KUKA KRL program: MyProgram_224().src

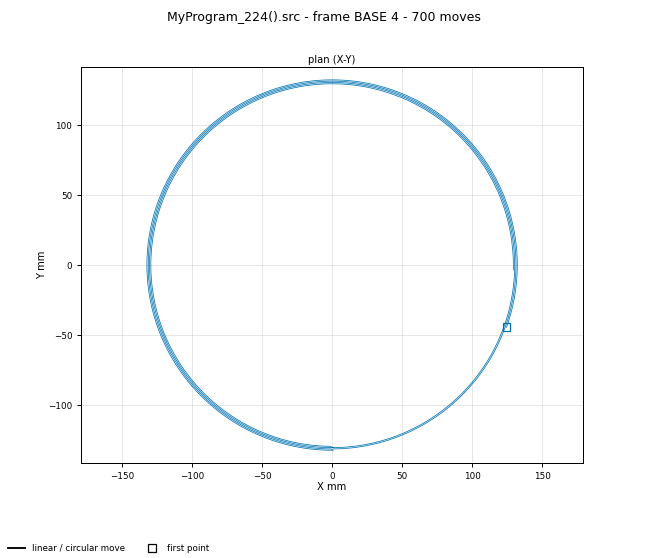
[picture p0: tool path of MyProgram_224().src in frame BASE 4, 700 of 700 moves have a stored position in this frame; points joined in program order, loops and branches not executed]
&ACCESS RVP
&REL 1
&PARAM TEMPLATE = C:\KRC\Roboter\Template\vorgabe
&PARAM EDITMASK = *
DEF MyProgram_224()
; ---- Setting reference (Base) ----
$BASE = BASE_DATA[4]

; --------------------------
; ---- Setting tool (TCP) ----
$TOOL = TOOL_DATA[3]
; --------------------------

$VEL.CP = VEL_APROX_PRINT
Startdeposition()
$VEL.CP = VEL_PRINT
LIN {X 124.5502,Y -44.5049,Z 155,A -21.604,B 21.391,C -0.8343,E1 21.5573,E2 829.1643} C_DIS
LIN {X 125.729,Y -41.0623,Z 155,A -19.4194,B 21.3896,C -0.8684,E1 21.5593,E2 826.9015} C_DIS
LIN {X 127.1456,Y -36.4403,Z 155,A -17.9667,B 21.3906,C -0.844,E1 21.5603,E2 825.525} C_DIS
LIN {X 127.8136,Y -34.0149,Z 155,A -16.9109,B 21.3905,C -0.8459,E1 21.5611,E2 824.4715} C_DIS
LIN {X 128.5807,Y -30.9894,Z 155,A -15.17,B 21.3896,C -0.8688,E1 21.5623,E2 822.6801} C_DIS
LIN {X 129.3697,Y -27.5135,Z 155,A -14.0813,B 21.3903,C -0.8518,E1 21.5629,E2 821.6452} C_DIS
LIN {X 129.9607,Y -24.5693,Z 155,A -12.5854,B 21.3897,C -0.8653,E1 21.5637,E2 820.123} C_DIS
LIN {X 130.7,Y -20.2702,Z 155,A -10.8405,B 21.3897,C -0.8643,E1 21.5645,E2 818.3928} C_DIS
LIN {X 131.174,Y -16.9359,Z 155,A -9.3618,B 21.3896,C -0.8699,E1 21.565,E2 816.9092} C_DIS
LIN {X 131.7113,Y -12.0763,Z 155,A -7.3959,B 21.3896,C -0.8694,E1 21.5656,E2 814.9586} C_DIS
LIN {X 132.0248,Y -7.9307,Z 155,A -5.4229,B 21.389,C -0.8834,E1 21.566,E2 812.9614} C_DIS
LIN {X 132.2116,Y -3.6774,Z 155,A -3.6274,B 21.3889,C -0.8869,E1 21.5662,E2 811.1688} C_DIS
LIN {X 132.263,Y 0.4651,Z 155,A -1.8131,B 21.3886,C -0.8936,E1 21.5662,E2 809.3493} C_DIS
LIN {X 132.2015,Y 4.0385,Z 155,A -0.2395,B 21.3884,C -0.8998,E1 21.5661,E2 807.7701} C_DIS
LIN {X 132.0289,Y 7.8652,Z 155,A 1.3524,B 21.3884,C -0.9018,E1 21.5659,E2 806.1838} C_DIS
LIN {X 131.7496,Y 11.6494,Z 155,A 3.0747,B 21.3879,C -0.9108,E1 21.5655,E2 804.4493} C_DIS
LIN {X 131.3233,Y 15.7351,Z 155,A 4.5909,B 21.3882,C -0.9038,E1 21.565,E2 802.9627} C_DIS
LIN {X 130.9162,Y 18.8242,Z 155,A 5.9988,B 21.3879,C -0.9108,E1 21.5645,E2 801.5455} C_DIS
LIN {X 130.4526,Y 21.8058,Z 155,A 7.3862,B 21.3876,C -0.9187,E1 21.5638,E2 800.1463} C_DIS
LIN {X 129.5637,Y 26.583,Z 155,A 10.6351,B 21.385,C -0.9803,E1 21.562,E2 796.7521} C_DIS
LIN {X 127.7263,Y 34.3422,Z 155,A 12.4336,B 21.3879,C -0.9114,E1 21.5609,E2 795.1537} C_DIS
LIN {X 126.694,Y 37.9805,Z 155,A 14.4558,B 21.387,C -0.9345,E1 21.5593,E2 793.0824} C_DIS
LIN {X 125.6249,Y 41.3749,Z 155,A 16.0763,B 21.3866,C -0.9428,E1 21.5578,E2 791.45} C_DIS
LIN {X 124.4093,Y 44.8959,Z 155,A 17.6313,B 21.3866,C -0.9448,E1 21.5564,E2 789.9} C_DIS
LIN {X 123.2107,Y 48.088,Z 155,A 19.0995,B 21.3864,C -0.9487,E1 21.5549,E2 788.4309} C_DIS
LIN {X 121.8494,Y 51.442,Z 155,A 20.6359,B 21.3862,C -0.9517,E1 21.5533,E2 786.8964} C_DIS
LIN {X 120.5815,Y 54.3464,Z 155,A 22.5754,B 21.3849,C -0.9825,E1 21.551,E2 784.8854} C_DIS
LIN {X 118.6107,Y 58.5216,Z 155,A 23.667,B 21.3865,C -0.9451,E1 21.5498,E2 783.9027} C_DIS
LIN {X 117.3355,Y 61.0402,Z 155,A 25.0814,B 21.386,C -0.9575,E1 21.548,E2 782.4636} C_DIS
LIN {X 115.8159,Y 63.8789,Z 155,A 26.7141,B 21.3854,C -0.9724,E1 21.5457,E2 780.8003} C_DIS
LIN {X 113.4513,Y 67.9904,Z 155,A 28.7424,B 21.3852,C -0.9767,E1 21.5429,E2 778.7729} C_DIS
LIN {X 111.1551,Y 71.6833,Z 155,A 30.6297,B 21.385,C -0.9817,E1 21.54,E2 776.8831} C_DIS
LIN {X 108.7622,Y 75.2641,Z 155,A 32.5525,B 21.3846,C -0.9892,E1 21.537,E2 774.9513} C_DIS
LIN {X 106.7868,Y 78.0415,Z 155,A 33.9503,B 21.3846,C -0.9892,E1 21.5347,E2 773.5616} C_DIS
LIN {X 104.1105,Y 81.5771,Z 155,A 36.6611,B 21.3827,C -1.031,E1 21.5299,E2 770.7518} C_DIS
LIN {X 99.9718,Y 86.6001,Z 155,A 38.3531,B 21.3848,C -0.9846,E1 21.5271,E2 769.1956} C_DIS
LIN {X 96.5456,Y 90.404,Z 155,A 40.8663,B 21.384,C -1.0033,E1 21.5223,E2 766.6446} C_DIS
LIN {X 93.4654,Y 93.5849,Z 155,A 42.7806,B 21.3838,C -1.0072,E1 21.5185,E2 764.7292} C_DIS
LIN {X 86.4701,Y 100.0837,Z 155,A 46.5284,B 21.3843,C -0.9976,E1 21.5109,E2 761.0258} C_DIS
LIN {X 83.7881,Y 102.3395,Z 155,A 48.3808,B 21.3834,C -1.0159,E1 21.5068,E2 759.132} C_DIS
LIN {X 80.2289,Y 105.1529,Z 155,A 50.3468,B 21.3833,C -1.0195,E1 21.5025,E2 757.1647} C_DIS
LIN {X 76.5729,Y 107.845,Z 155,A 52.3369,B 21.3831,C -1.024,E1 21.498,E2 755.1707} C_DIS
LIN {X 72.8868,Y 110.3692,Z 155,A 54.236,B 21.383,C -1.0255,E1 21.4936,E2 753.2751} C_DIS
LIN {X 68.9512,Y 112.8698,Z 155,A 56.2434,B 21.3829,C -1.028,E1 21.4888,E2 751.2683} C_DIS
LIN {X 64.7177,Y 115.3492,Z 155,A 58.3316,B 21.3829,C -1.0294,E1 21.4838,E2 749.1838} C_DIS
LIN {X 60.9874,Y 117.3632,Z 155,A 60.4088,B 21.3822,C -1.0429,E1 21.4786,E2 747.0768} C_DIS
LIN {X 57.9889,Y 118.8735,Z 155,A 61.7981,B 21.3822,C -1.0417,E1 21.4751,E2 745.695} C_DIS
LIN {X 53.656,Y 120.8903,Z 155,A 63.5823,B 21.3827,C -1.0312,E1 21.4707,E2 743.9449} C_DIS
LIN {X 51.011,Y 122.0294,Z 155,A 64.8174,B 21.3827,C -1.032,E1 21.4675,E2 742.7111} C_DIS
LIN {X 47.2563,Y 123.534,Z 155,A 66.535,B 21.3827,C -1.0322,E1 21.463,E2 740.9976} C_DIS
LIN {X 43.2481,Y 124.9917,Z 155,A 68.4763,B 21.3824,C -1.0381,E1 21.4579,E2 739.0447} C_DIS
LIN {X 39.7093,Y 126.1618,Z 155,A 70.0332,B 21.3824,C -1.0368,E1 21.4538,E2 737.4948} C_DIS
LIN {X 33.5194,Y 127.9458,Z 155,A 73.1745,B 21.3816,C -1.0545,E1 21.4452,E2 734.3114} C_DIS
LIN {X 30.1368,Y 128.7851,Z 155,A 74.2876,B 21.3824,C -1.0376,E1 21.4423,E2 733.2463} C_DIS
LIN {X 26.5128,Y 129.578,Z 155,A 75.9495,B 21.3823,C -1.0409,E1 21.4378,E2 731.578} C_DIS
LIN {X 23.2374,Y 130.2052,Z 155,A 77.392,B 21.3823,C -1.0414,E1 21.4338,E2 730.136} C_DIS
LIN {X 19.5153,Y 130.8169,Z 155,A 79.2255,B 21.3818,C -1.0507,E1 21.4287,E2 728.2789} C_DIS
LIN {X 15.5547,Y 131.3448,Z 155,A 80.7732,B 21.3822,C -1.0431,E1 21.4245,E2 726.7537} C_DIS
LIN {X 11.8097,Y 131.7361,Z 155,A 82.5091,B 21.382,C -1.0479,E1 21.4196,E2 725.0059} C_DIS
LIN {X 7.9894,Y 132.0212,Z 155,A 84.0684,B 21.3822,C -1.0436,E1 21.4153,E2 723.4592} C_DIS
LIN {X 3.5658,Y 132.2147,Z 155,A 85.9886,B 21.3822,C -1.0436,E1 21.4099,E2 721.5397} C_DIS
LIN {X -0.6478,Y 132.2612,Z 155,A 87.8269,B 21.3822,C -1.0439,E1 21.4048,E2 719.7007} C_DIS
LIN {X -4.8887,Y 132.1726,Z 155,A 89.6565,B 21.3822,C -1.0431,E1 21.3997,E2 717.873} C_DIS
LIN {X -8.5001,Y 131.9898,Z 155,A 91.3658,B 21.3819,C -1.0488,E1 21.3949,E2 716.1475} C_DIS
LIN {X -13.2402,Y 131.5996,Z 155,A 93.3984,B 21.382,C -1.0466,E1 21.3893,E2 714.1196} C_DIS
LIN {X -17.2614,Y 131.1314,Z 155,A 95.0131,B 21.3823,C -1.0396,E1 21.3848,E2 712.5227} C_DIS
LIN {X -21.0472,Y 130.5792,Z 155,A 97.0435,B 21.3816,C -1.0547,E1 21.3791,E2 710.4488} C_DIS
LIN {X -24.4702,Y 129.9796,Z 155,A 98,B 21.3828,C -1.0299,E1 21.3767,E2 709.5592} C_DIS
LIN {X -26.9614,Y 129.4867,Z 155,A 100.1971,B 21.3806,C -1.0765,E1 21.3703,E2 707.231} C_DIS
LIN {X -33.2052,Y 128.0282,Z 155,A 102.0517,B 21.3826,C -1.0339,E1 21.3656,E2 705.4902} C_DIS
LIN {X -38.8586,Y 126.4253,Z 155,A 104.581,B 21.3828,C -1.0306,E1 21.3588,E2 702.9652} C_DIS
LIN {X -41.9806,Y 125.4232,Z 155,A 106.0925,B 21.3827,C -1.0328,E1 21.3548,E2 701.4443} C_DIS
LIN {X -45.4039,Y 124.2261,Z 155,A 107.7019,B 21.3827,C -1.0325,E1 21.3505,E2 699.8319} C_DIS
LIN {X -54.3042,Y 120.6004,Z 155,A 111.6937,B 21.3833,C -1.0194,E1 21.3403,E2 695.8653} C_DIS
LIN {X -56.8154,Y 119.4376,Z 155,A 113.5157,B 21.3821,C -1.0441,E1 21.3355,E2 693.97} C_DIS
LIN {X -60.8021,Y 117.4605,Z 155,A 115.0137,B 21.3831,C -1.0227,E1 21.3319,E2 692.526} C_DIS
LIN {X -64.4819,Y 115.4817,Z 155,A 116.8834,B 21.3831,C -1.0222,E1 21.3274,E2 690.6514} C_DIS
LIN {X -68.3799,Y 113.2166,Z 155,A 118.7978,B 21.3834,C -1.0171,E1 21.3228,E2 688.744} C_DIS
LIN {X -72.1535,Y 110.8499,Z 155,A 120.7581,B 21.3834,C -1.0149,E1 21.3182,E2 686.7825} C_DIS
LIN {X -75.9078,Y 108.3142,Z 155,A 122.7343,B 21.3836,C -1.0116,E1 21.3136,E2 684.8073} C_DIS
LIN {X -79.3536,Y 105.8157,Z 155,A 124.6149,B 21.3837,C -1.0094,E1 21.3094,E2 682.9248} C_DIS
LIN {X -82.9748,Y 102.9999,Z 155,A 126.5719,B 21.384,C -1.004,E1 21.3051,E2 680.9742} C_DIS
LIN {X -86.4303,Y 100.118,Z 155,A 128.5306,B 21.3841,C -1.0001,E1 21.3009,E2 679.017} C_DIS
LIN {X -89.4659,Y 97.4148,Z 155,A 130.2762,B 21.3843,C -0.9955,E1 21.2973,E2 677.2759} C_DIS
LIN {X -92.5632,Y 94.4767,Z 155,A 132.184,B 21.3844,C -0.9936,E1 21.2935,E2 675.3638} C_DIS
LIN {X -95.8388,Y 91.1527,Z 155,A 134.2016,B 21.3846,C -0.9886,E1 21.2896,E2 673.3497} C_DIS
LIN {X -98.8107,Y 87.9227,Z 155,A 136.1481,B 21.3848,C -0.9858,E1 21.2859,E2 671.4007} C_DIS
LIN {X -101.7408,Y 84.5141,Z 155,A 138.0878,B 21.385,C -0.9805,E1 21.2825,E2 669.4649} C_DIS
LIN {X -104.624,Y 80.9174,Z 155,A 140.0687,B 21.3853,C -0.9746,E1 21.279,E2 667.4892} C_DIS
LIN {X -107.2983,Y 77.3369,Z 155,A 142.0449,B 21.3854,C -0.9711,E1 21.2758,E2 665.5112} C_DIS
LIN {X -109.7964,Y 73.7475,Z 155,A 143.9683,B 21.3856,C -0.9672,E1 21.2727,E2 663.5874} C_DIS
LIN {X -112.3661,Y 69.7687,Z 155,A 145.9858,B 21.3859,C -0.9601,E1 21.2697,E2 661.5774} C_DIS
LIN {X -114.6205,Y 66.0003,Z 155,A 147.9225,B 21.3861,C -0.9561,E1 21.267,E2 659.6397} C_DIS
LIN {X -116.7267,Y 62.1995,Z 155,A 149.701,B 21.3865,C -0.9464,E1 21.2646,E2 657.8766} C_DIS
LIN {X -117.9148,Y 59.9115,Z 155,A 150.9475,B 21.3864,C -0.9485,E1 21.263,E2 656.6165} C_DIS
LIN {X -120.222,Y 55.1373,Z 155,A 153.133,B 21.3869,C -0.9371,E1 21.2605,E2 654.4481} C_DIS
LIN {X -121.558,Y 52.1257,Z 155,A 154.7052,B 21.3868,C -0.9388,E1 21.2587,E2 652.8611} C_DIS
LIN {X -123.1922,Y 48.1356,Z 155,A 156.52,B 21.3871,C -0.931,E1 21.2568,E2 651.0557} C_DIS
LIN {X -124.4083,Y 44.8986,Z 155,A 157.9622,B 21.3874,C -0.9242,E1 21.2554,E2 649.6227} C_DIS
LIN {X -125.4654,Y 41.8539,Z 155,A 159.3937,B 21.3875,C -0.9213,E1 21.2541,E2 648.1894} C_DIS
LIN {X -126.4976,Y 38.6223,Z 155,A 160.9052,B 21.3876,C -0.9185,E1 21.2529,E2 646.6753} C_DIS
LIN {X -127.4238,Y 35.4478,Z 155,A 162.2798,B 21.3879,C -0.9117,E1 21.2518,E2 645.3101} C_DIS
LIN {X -128.2741,Y 32.2364,Z 155,A 163.7978,B 21.3879,C -0.9104,E1 21.2508,E2 643.7851} C_DIS
LIN {X -129.0531,Y 28.9638,Z 155,A 165.2081,B 21.3882,C -0.9039,E1 21.2499,E2 642.3829} C_DIS
LIN {X -129.8053,Y 25.3821,Z 155,A 167.4969,B 21.3873,C -0.9276,E1 21.2486,E2 640.0123} C_DIS
LIN {X -130.6773,Y 20.4172,Z 155,A 168.7767,B 21.389,C -0.8838,E1 21.2481,E2 638.8446} C_DIS
LIN {X -130.9951,Y 18.272,Z 155,A 170.1588,B 21.3884,C -0.8988,E1 21.2475,E2 637.4113} C_DIS
LIN {X -131.5768,Y 13.4684,Z 155,A 172.05,B 21.389,C -0.8837,E1 21.247,E2 635.5481} C_DIS
LIN {X -131.8362,Y 10.6247,Z 155,A 173.2818,B 21.3892,C -0.8796,E1 21.2467,E2 634.319} C_DIS
LIN {X -132.0466,Y 7.5773,Z 155,A 174.7987,B 21.389,C -0.8832,E1 21.2464,E2 632.781} C_DIS
LIN {X -132.2186,Y 3.4248,Z 155,A 176.7444,B 21.389,C -0.8835,E1 21.2462,E2 630.8209} C_DIS
LIN {X -132.2512,Y -1.7936,Z 155,A 179.233,B 21.389,C -0.8856,E1 21.2462,E2 628.3084} C_DIS
LIN {X -132.1309,Y -5.9428,Z 155,A -179.4763,B 21.39,C -0.8591,E1 21.2464,E2 627.0817} C_DIS
LIN {X -131.5695,Y -13.5366,Z 155,A -176.183,B 21.3904,C -0.8484,E1 21.2472,E2 623.7943} C_DIS
LIN {X -131.2466,Y -16.3729,Z 155,A -174.3698,B 21.3896,C -0.8681,E1 21.2478,E2 621.9136} C_DIS
LIN {X -130.6806,Y -20.3954,Z 155,A -173.0766,B 21.3906,C -0.8435,E1 21.2483,E2 620.6794} C_DIS
LIN {X -129.8727,Y -25.0297,Z 155,A -170.9993,B 21.3907,C -0.8388,E1 21.2493,E2 618.6004} C_DIS
LIN {X -129.0995,Y -28.7605,Z 155,A -169.2149,B 21.3907,C -0.8392,E1 21.2504,E2 616.8025} C_DIS
LIN {X -128.1718,Y -32.6393,Z 155,A -167.6177,B 21.3911,C -0.8286,E1 21.2515,E2 615.2233} C_DIS
LIN {X -127.3439,Y -35.7334,Z 155,A -166.1625,B 21.3911,C -0.8272,E1 21.2525,E2 613.7619} C_DIS
LIN {X -126.1004,Y -39.9017,Z 155,A -164.2744,B 21.3914,C -0.8217,E1 21.2541,E2 611.8761} C_DIS
LIN {X -124.9391,Y -43.3996,Z 155,A -162.0517,B 21.3906,C -0.8429,E1 21.2562,E2 609.5798} C_DIS
LIN {X -123.1721,Y -48.1873,Z 155,A -160.5089,B 21.3919,C -0.8088,E1 21.2577,E2 608.1209} C_DIS
LIN {X -122.0171,Y -51.0404,Z 155,A -159.1547,B 21.3919,C -0.8058,E1 21.2591,E2 606.7659} C_DIS
LIN {X -119.9799,Y -55.6609,Z 155,A -156.9065,B 21.3921,C -0.8021,E1 21.2617,E2 604.5132} C_DIS
LIN {X -118.4929,Y -58.7605,Z 155,A -155.4227,B 21.3922,C -0.7977,E1 21.2635,E2 603.0319} C_DIS
LIN {X -116.456,Y -62.7042,Z 155,A -153.164,B 21.3919,C -0.8064,E1 21.2665,E2 600.735} C_DIS
LIN {X -114.7788,Y -65.7242,Z 155,A -152.0955,B 21.3927,C -0.7846,E1 21.2679,E2 599.72} C_DIS
LIN {X -112.9693,Y -68.7889,Z 155,A -150.3322,B 21.3925,C -0.7898,E1 21.2705,E2 597.9317} C_DIS
LIN {X -110.1869,Y -73.1625,Z 155,A -148.1067,B 21.3928,C -0.7831,E1 21.2738,E2 595.7111} C_DIS
LIN {X -107.807,Y -76.6263,Z 155,A -146.2215,B 21.3928,C -0.7813,E1 21.2769,E2 593.8199} C_DIS
LIN {X -105.1788,Y -80.195,Z 155,A -144.3652,B 21.3931,C -0.774,E1 21.28,E2 591.9732} C_DIS
LIN {X -102.7283,Y -83.3115,Z 155,A -142.5551,B 21.3931,C -0.7738,E1 21.2831,E2 590.1536} C_DIS
LIN {X -99.7992,Y -86.7984,Z 155,A -140.5967,B 21.3933,C -0.7686,E1 21.2867,E2 588.1987} C_DIS
LIN {X -97.04,Y -89.873,Z 155,A -138.787,B 21.3933,C -0.7655,E1 21.2901,E2 586.3881} C_DIS
LIN {X -93.9839,Y -93.0638,Z 155,A -136.8822,B 21.3935,C -0.761,E1 21.2938,E2 584.486} C_DIS
LIN {X -90.7189,Y -96.249,Z 155,A -134.9164,B 21.3937,C -0.7565,E1 21.2978,E2 582.5229} C_DIS
LIN {X -87.4611,Y -99.2189,Z 155,A -132.9959,B 21.3937,C -0.7532,E1 21.3018,E2 580.6024} C_DIS
LIN {X -84.2512,Y -101.9585,Z 155,A -131.2006,B 21.3939,C -0.7483,E1 21.3056,E2 578.8123} C_DIS
LIN {X -81.0487,Y -104.5223,Z 155,A -129.3602,B 21.3939,C -0.7478,E1 21.3096,E2 576.9653} C_DIS
LIN {X -77.4558,Y -107.2121,Z 155,A -127.511,B 21.3942,C -0.7404,E1 21.3138,E2 575.1288} C_DIS
LIN {X -74.3148,Y -109.4127,Z 155,A -125.7307,B 21.3942,C -0.7427,E1 21.3179,E2 573.3348} C_DIS
LIN {X -70.4361,Y -111.949,Z 155,A -123.6302,B 21.3942,C -0.7436,E1 21.3229,E2 571.2239} C_DIS
LIN {X -66.089,Y -114.5691,Z 155,A -121.5245,B 21.3943,C -0.7364,E1 21.3279,E2 569.1304} C_DIS
LIN {X -61.3781,Y -117.1581,Z 155,A -119.659,B 21.3951,C -0.7134,E1 21.3323,E2 567.322} C_DIS
LIN {X -58.57,Y -118.5868,Z 155,A -117.835,B 21.3945,C -0.7314,E1 21.337,E2 565.4426} C_DIS
LIN {X -54.8925,Y -120.3352,Z 155,A -116.0091,B 21.3945,C -0.732,E1 21.3417,E2 563.6096} C_DIS
LIN {X -50.3246,Y -122.3161,Z 155,A -114.0237,B 21.3948,C -0.7223,E1 21.3467,E2 561.6456} C_DIS
LIN {X -47.842,Y -123.3063,Z 155,A -112.837,B 21.3948,C -0.7224,E1 21.3498,E2 560.4554} C_DIS
LIN {X -44.4521,Y -124.5693,Z 155,A -111.2706,B 21.3948,C -0.721,E1 21.3539,E2 558.8893} C_DIS
LIN {X -41.2506,Y -125.6663,Z 155,A -109.311,B 21.3942,C -0.7414,E1 21.3593,E2 556.8691} C_DIS
LIN {X -37.3729,Y -126.8725,Z 155,A -108.2622,B 21.3952,C -0.709,E1 21.3618,E2 555.9074} C_DIS
LIN {X -33.4908,Y -127.9534,Z 155,A -106.3297,B 21.395,C -0.716,E1 21.3671,E2 553.9521} C_DIS
LIN {X -30.237,Y -128.762,Z 155,A -104.8357,B 21.395,C -0.717,E1 21.3712,E2 552.4529} C_DIS
LIN {X -26.2904,Y -129.6232,Z 155,A -103.0513,B 21.395,C -0.7177,E1 21.3761,E2 550.6639} C_DIS
LIN {X -22.2489,Y -130.3787,Z 155,A -101.0192,B 21.3946,C -0.7282,E1 21.3817,E2 548.6006} C_DIS
LIN {X -18.1653,Y -131.0103,Z 155,A -99.5497,B 21.3951,C -0.7135,E1 21.3857,E2 547.17} C_DIS
LIN {X -15.2291,Y -131.3836,Z 155,A -98.0773,B 21.3948,C -0.7217,E1 21.3898,E2 545.6739} C_DIS
LIN {X -11.1489,Y -131.7919,Z 155,A -96.4452,B 21.395,C -0.7151,E1 21.3943,E2 544.0589} C_DIS
LIN {X -7.5628,Y -132.0475,Z 155,A -94.7511,B 21.3948,C -0.7212,E1 21.3991,E2 542.3474} C_DIS
LIN {X -3.6165,Y -132.2133,Z 155,A -93.1246,B 21.395,C -0.7176,E1 21.4036,E2 540.7305} C_DIS
LIN {X 0.935,Y -132.2575,Z 155,A -91.318,B 21.3952,C -0.7106,E1 21.4086,E2 538.9431} C_DIS
Enddeposition()
LIN {X 0.935,Y -132.2575,Z 155,A -91.318,B 21.3952,C -0.7106,E1 21.4086,E2 538.9431} C_DIS
Startdeposition()
$VEL.CP = VEL_PRINT
LIN {X -0.4574,Y -131.327,Z 155,A -92.2415,B 20.3181,C -0.5393,E1 20.3234,E2 540.2372} C_DIS
LIN {X -4.5745,Y -131.2488,Z 155,A -93.9797,B 20.318,C -0.5415,E1 20.3186,E2 541.9693} C_DIS
LIN {X -8.3286,Y -131.0633,Z 155,A -95.6611,B 20.318,C -0.5398,E1 20.3139,E2 543.6563} C_DIS
LIN {X -12.4961,Y -130.7315,Z 155,A -97.4007,B 20.318,C -0.5435,E1 20.3091,E2 545.3864} C_DIS
LIN {X -16.2524,Y -130.3196,Z 155,A -98.9995,B 20.3179,C -0.5458,E1 20.3047,E2 546.9799} C_DIS
LIN {X -22.3313,Y -129.4167,Z 155,A -101.8626,B 20.3181,C -0.5391,E1 20.2967,E2 549.8655} C_DIS
LIN {X -26.189,Y -128.6894,Z 155,A -103.46,B 20.3179,C -0.5445,E1 20.2924,E2 551.4493} C_DIS
LIN {X -29.7977,Y -127.9032,Z 155,A -105.036,B 20.3179,C -0.5468,E1 20.2881,E2 553.0214} C_DIS
LIN {X -33.2063,Y -127.0613,Z 155,A -106.7097,B 20.3179,C -0.5419,E1 20.2835,E2 554.7122} C_DIS
LIN {X -36.7118,Y -126.0916,Z 155,A -108.2274,B 20.3179,C -0.5458,E1 20.2794,E2 556.2217} C_DIS
LIN {X -40.9923,Y -124.7666,Z 155,A -110.1763,B 20.3179,C -0.5475,E1 20.2743,E2 558.1699} C_DIS
LIN {X -44.5325,Y -123.5461,Z 155,A -111.758,B 20.3178,C -0.5511,E1 20.2701,E2 559.7453} C_DIS
LIN {X -47.5952,Y -122.3988,Z 155,A -113.1591,B 20.3177,C -0.5534,E1 20.2665,E2 561.1432} C_DIS
LIN {X -52.94,Y -120.186,Z 155,A -115.8716,B 20.3178,C -0.5485,E1 20.2594,E2 563.878} C_DIS
LIN {X -56.2415,Y -118.6752,Z 155,A -117.363,B 20.3177,C -0.554,E1 20.2557,E2 565.3579} C_DIS
LIN {X -59.3741,Y -117.1388,Z 155,A -118.8163,B 20.3176,C -0.5587,E1 20.2521,E2 566.8027} C_DIS
LIN {X -62.2428,Y -115.6421,Z 155,A -120.349,B 20.3176,C -0.5557,E1 20.2483,E2 568.3494} C_DIS
LIN {X -66.1322,Y -113.4635,Z 155,A -122.1088,B 20.3174,C -0.5657,E1 20.244,E2 570.0865} C_DIS
LIN {X -70.863,Y -110.5699,Z 155,A -124.7407,B 20.3174,C -0.5609,E1 20.2377,E2 572.7428} C_DIS
LIN {X -74.647,Y -108.052,Z 155,A -126.9007,B 20.3176,C -0.5571,E1 20.2327,E2 574.9229} C_DIS
LIN {X -78.7735,Y -105.0817,Z 155,A -129.0136,B 20.3174,C -0.5651,E1 20.228,E2 577.0222} C_DIS
LIN {X -82.2617,Y -102.3734,Z 155,A -130.9141,B 20.3173,C -0.5696,E1 20.2238,E2 578.9184} C_DIS
LIN {X -85.6766,Y -99.5328,Z 155,A -132.8098,B 20.3171,C -0.5749,E1 20.2198,E2 580.808} C_DIS
LIN {X -88.7478,Y -96.8045,Z 155,A -134.4497,B 20.3169,C -0.5844,E1 20.2164,E2 582.4286} C_DIS
LIN {X -91.2698,Y -94.4304,Z 155,A -136.1491,B 20.3169,C -0.5801,E1 20.2129,E2 584.1492} C_DIS
LIN {X -94.2318,Y -91.4749,Z 155,A -138.0169,B 20.3169,C -0.5823,E1 20.2093,E2 586.0206} C_DIS
LIN {X -97.334,Y -88.1667,Z 155,A -139.9431,B 20.3167,C -0.5887,E1 20.2056,E2 587.939} C_DIS
LIN {X -100.131,Y -84.9768,Z 155,A -141.6544,B 20.3165,C -0.5983,E1 20.2025,E2 589.6323} C_DIS
LIN {X -102.5896,Y -81.9921,Z 155,A -143.5741,B 20.3166,C -0.5932,E1 20.1991,E2 591.578} C_DIS
LIN {X -105.2683,Y -78.523,Z 155,A -145.5059,B 20.3166,C -0.5971,E1 20.1959,E2 593.5103} C_DIS
LIN {X -107.7885,Y -75.0261,Z 155,A -147.3519,B 20.3163,C -0.603,E1 20.1929,E2 595.3505} C_DIS
LIN {X -109.3735,Y -72.6965,Z 155,A -149.1542,B 20.3169,C -0.5842,E1 20.19,E2 597.2186} C_DIS
LIN {X -112.038,Y -68.5185,Z 155,A -151.7095,B 20.3171,C -0.575,E1 20.1862,E2 599.8172} C_DIS
LIN {X -115.4851,Y -62.535,Z 155,A -153.8543,B 20.316,C -0.6159,E1 20.1835,E2 601.8577} C_DIS
LIN {X -117.5664,Y -58.5245,Z 155,A -155.7607,B 20.3157,C -0.6238,E1 20.1811,E2 603.7541} C_DIS
LIN {X -118.9455,Y -55.6696,Z 155,A -157.3837,B 20.3159,C -0.6185,E1 20.1791,E2 605.4036} C_DIS
LIN {X -121.0737,Y -50.8724,Z 155,A -159.1859,B 20.3151,C -0.6435,E1 20.1772,E2 607.1457} C_DIS
LIN {X -122.0831,Y -48.4031,Z 155,A -161.437,B 20.3163,C -0.6057,E1 20.1748,E2 609.5224} C_DIS
LIN {X -124.166,Y -42.7744,Z 155,A -163.2677,B 20.3152,C -0.643,E1 20.1731,E2 611.2581} C_DIS
LIN {X -125.4699,Y -38.7846,Z 155,A -165.0573,B 20.315,C -0.6499,E1 20.1716,E2 613.0403} C_DIS
LIN {X -126.3897,Y -35.6727,Z 155,A -166.5112,B 20.3149,C -0.6527,E1 20.1705,E2 614.4968} C_DIS
LIN {X -127.2775,Y -32.3611,Z 155,A -168.0169,B 20.3147,C -0.6568,E1 20.1694,E2 616.0016} C_DIS
LIN {X -128.2074,Y -28.4651,Z 155,A -169.8659,B 20.3147,C -0.6583,E1 20.1683,E2 617.8601} C_DIS
LIN {X -128.9707,Y -24.7668,Z 155,A -171.486,B 20.3145,C -0.6644,E1 20.1674,E2 619.4746} C_DIS
LIN {X -129.6905,Y -20.6776,Z 155,A -173.2236,B 20.3142,C -0.6727,E1 20.1666,E2 621.201} C_DIS
LIN {X -130.5086,Y -14.6534,Z 155,A -176.7611,B 20.315,C -0.6479,E1 20.1654,E2 624.8373} C_DIS
LIN {X -131.0403,Y -8.7014,Z 155,A -178.4614,B 20.3137,C -0.6899,E1 20.165,E2 626.4285} C_DIS
LIN {X -131.3021,Y -2.5869,Z 155,A 178.7707,B 20.3135,C -0.6946,E1 20.1647,E2 629.2038} C_DIS
LIN {X -131.2061,Y 5.6711,Z 155,A 175.0184,B 20.3134,C -0.7003,E1 20.1649,E2 632.9681} C_DIS
LIN {X -131.044,Y 8.6415,Z 155,A 173.4875,B 20.3135,C -0.6956,E1 20.1652,E2 634.524} C_DIS
LIN {X -130.7792,Y 11.9986,Z 155,A 171.8414,B 20.3135,C -0.6937,E1 20.1656,E2 636.1884} C_DIS
LIN {X -130.3238,Y 16.2171,Z 155,A 170.348,B 20.3129,C -0.7129,E1 20.1661,E2 637.6373} C_DIS
LIN {X -129.6592,Y 20.8774,Z 155,A 168.1766,B 20.3129,C -0.7149,E1 20.167,E2 639.8191} C_DIS
LIN {X -128.8296,Y 25.5001,Z 155,A 166.2068,B 20.3125,C -0.7243,E1 20.168,E2 641.7764} C_DIS
LIN {X -128.0241,Y 29.2685,Z 155,A 164.7344,B 20.3121,C -0.7374,E1 20.1689,E2 643.2217} C_DIS
LIN {X -127.3118,Y 32.2259,Z 155,A 163.3107,B 20.3121,C -0.7379,E1 20.1699,E2 644.6546} C_DIS
LIN {X -126.4437,Y 35.4796,Z 155,A 161.8687,B 20.3119,C -0.7434,E1 20.1709,E2 646.091} C_DIS
LIN {X -125.6223,Y 38.2866,Z 155,A 160.4672,B 20.3119,C -0.7426,E1 20.1721,E2 647.505} C_DIS
LIN {X -124.3647,Y 42.1992,Z 155,A 158.593,B 20.3119,C -0.745,E1 20.1737,E2 649.3859} C_DIS
LIN {X -123.0982,Y 45.7572,Z 155,A 157.1587,B 20.3114,C -0.758,E1 20.175,E2 650.7926} C_DIS
LIN {X -121.9194,Y 48.811,Z 155,A 155.6151,B 20.3114,C -0.758,E1 20.1766,E2 652.3473} C_DIS
LIN {X -120.4881,Y 52.2437,Z 155,A 154.0251,B 20.3112,C -0.764,E1 20.1784,E2 653.9309} C_DIS
LIN {X -119.3897,Y 54.7088,Z 155,A 152.0252,B 20.3121,C -0.7366,E1 20.1808,E2 656.0239} C_DIS
LIN {X -116.9344,Y 59.7758,Z 155,A 150.3334,B 20.3108,C -0.7723,E1 20.1828,E2 657.6236} C_DIS
LIN {X -115.3316,Y 62.8164,Z 155,A 148.7131,B 20.3108,C -0.772,E1 20.185,E2 659.2556} C_DIS
LIN {X -113.1196,Y 66.7178,Z 155,A 146.8595,B 20.3105,C -0.7814,E1 20.1875,E2 661.0941} C_DIS
LIN {X -110.7182,Y 70.6314,Z 155,A 144.7852,B 20.3105,C -0.7842,E1 20.1906,E2 663.1736} C_DIS
LIN {X -108.528,Y 73.9534,Z 155,A 142.9536,B 20.3104,C -0.7853,E1 20.1935,E2 665.0136} C_DIS
LIN {X -106.02,Y 77.5055,Z 155,A 141.0459,B 20.3102,C -0.7899,E1 20.1966,E2 666.9196} C_DIS
LIN {X -103.3717,Y 81.0036,Z 155,A 139.1526,B 20.31,C -0.7957,E1 20.1998,E2 668.8075} C_DIS
LIN {X -100.5253,Y 84.51,Z 155,A 137.1987,B 20.3098,C -0.8013,E1 20.2032,E2 670.7565} C_DIS
LIN {X -97.6265,Y 87.8431,Z 155,A 135.2783,B 20.3096,C -0.8063,E1 20.2068,E2 672.6733} C_DIS
LIN {X -94.7362,Y 90.9528,Z 155,A 133.4091,B 20.3094,C -0.8101,E1 20.2104,E2 674.5418} C_DIS
LIN {X -91.7217,Y 93.992,Z 155,A 131.4976,B 20.3094,C -0.8128,E1 20.2142,E2 676.4557} C_DIS
LIN {X -88.6894,Y 96.8582,Z 155,A 129.6751,B 20.3092,C -0.8168,E1 20.2179,E2 678.2759} C_DIS
LIN {X -85.597,Y 99.6014,Z 155,A 127.8715,B 20.309,C -0.8207,E1 20.2217,E2 680.0769} C_DIS
LIN {X -82.1751,Y 102.4433,Z 155,A 125.87,B 20.309,C -0.8225,E1 20.226,E2 682.0829} C_DIS
LIN {X -78.7042,Y 105.1333,Z 155,A 123.9224,B 20.3089,C -0.8252,E1 20.2303,E2 684.0316} C_DIS
LIN {X -75.1503,Y 107.702,Z 155,A 122.098,B 20.3086,C -0.8323,E1 20.2345,E2 685.8433} C_DIS
LIN {X -72.1057,Y 109.7636,Z 155,A 120.4113,B 20.3086,C -0.8321,E1 20.2384,E2 687.5375} C_DIS
LIN {X -68.4407,Y 112.0857,Z 155,A 118.5165,B 20.3085,C -0.8354,E1 20.2429,E2 689.4303} C_DIS
LIN {X -64.6974,Y 114.2877,Z 155,A 116.5881,B 20.3084,C -0.8374,E1 20.2475,E2 691.3603} C_DIS
LIN {X -61.9533,Y 115.7977,Z 155,A 115.1497,B 20.3084,C -0.8368,E1 20.2511,E2 692.8055} C_DIS
LIN {X -57.3218,Y 118.1591,Z 155,A 113.0027,B 20.3081,C -0.845,E1 20.2564,E2 694.9359} C_DIS
LIN {X -54.8399,Y 119.3291,Z 155,A 111.529,B 20.3084,C -0.836,E1 20.2602,E2 696.4402} C_DIS
LIN {X -51.7437,Y 120.7035,Z 155,A 109.8015,B 20.3087,C -0.8283,E1 20.2647,E2 698.195} C_DIS
LIN {X -47.4141,Y 122.4692,Z 155,A 108.3214,B 20.3078,C -0.8528,E1 20.2684,E2 699.6083} C_DIS
LIN {X -43.6857,Y 123.8501,Z 155,A 106.5195,B 20.3078,C -0.8522,E1 20.2732,E2 701.4163} C_DIS
LIN {X -40.2306,Y 125.0135,Z 155,A 104.9636,B 20.3077,C -0.8554,E1 20.2773,E2 702.9666} C_DIS
LIN {X -35.9521,Y 126.3116,Z 155,A 103.0212,B 20.3076,C -0.8578,E1 20.2825,E2 704.9064} C_DIS
LIN {X -33.4255,Y 127.0029,Z 155,A 101.1597,B 20.3087,C -0.8305,E1 20.2878,E2 706.85} C_DIS
LIN {X -28.1111,Y 128.2838,Z 155,A 99.6107,B 20.3072,C -0.8656,E1 20.2917,E2 708.3002} C_DIS
LIN {X -20.8749,Y 129.6597,Z 155,A 96.154,B 20.3076,C -0.8581,E1 20.3013,E2 711.783} C_DIS
LIN {X -16.9131,Y 130.2337,Z 155,A 94.639,B 20.3071,C -0.8684,E1 20.3054,E2 713.2698} C_DIS
LIN {X -12.6923,Y 130.7126,Z 155,A 92.2348,B 20.308,C -0.8472,E1 20.3122,E2 715.7368} C_DIS
LIN {X -8.6348,Y 131.0444,Z 155,A 90.8278,B 20.3074,C -0.8626,E1 20.316,E2 717.1} C_DIS
LIN {X -4.8757,Y 131.2371,Z 155,A 89.183,B 20.3074,C -0.863,E1 20.3206,E2 718.7442} C_DIS
LIN {X -0.8549,Y 131.3247,Z 155,A 87.4879,B 20.3072,C -0.8658,E1 20.3253,E2 720.4314} C_DIS
LIN {X 2.6849,Y 131.301,Z 155,A 85.6692,B 20.3077,C -0.8548,E1 20.3305,E2 722.2814} C_DIS
LIN {X 5.934,Y 131.1949,Z 155,A 84.4582,B 20.3073,C -0.8632,E1 20.3338,E2 723.4677} C_DIS
LIN {X 9.8062,Y 130.961,Z 155,A 82.8237,B 20.3073,C -0.8655,E1 20.3383,E2 725.0947} C_DIS
LIN {X 13.4666,Y 130.6364,Z 155,A 81.0789,B 20.3075,C -0.8595,E1 20.3432,E2 726.8555} C_DIS
LIN {X 19.5197,Y 129.8698,Z 155,A 78.5117,B 20.3074,C -0.8626,E1 20.3503,E2 729.4109} C_DIS
LIN {X 23.1004,Y 129.2796,Z 155,A 76.9981,B 20.3073,C -0.8649,E1 20.3544,E2 730.9159} C_DIS
LIN {X 26.3341,Y 128.6599,Z 155,A 75.6163,B 20.3073,C -0.8665,E1 20.3582,E2 732.2911} C_DIS
LIN {X 28.9455,Y 128.0979,Z 155,A 74.2778,B 20.3075,C -0.8587,E1 20.3619,E2 733.6496} C_DIS
LIN {X 33.4926,Y 126.985,Z 155,A 72.2433,B 20.3075,C -0.8577,E1 20.3674,E2 735.683} C_DIS
LIN {X 37.9774,Y 125.7169,Z 155,A 70.3086,B 20.3075,C -0.8603,E1 20.3725,E2 737.6061} C_DIS
LIN {X 41.5191,Y 124.5911,Z 155,A 68.6993,B 20.3075,C -0.8595,E1 20.3768,E2 739.2139} C_DIS
LIN {X 45.2028,Y 123.3044,Z 155,A 67.0882,B 20.3075,C -0.8617,E1 20.381,E2 740.8145} C_DIS
LIN {X 49.9445,Y 121.4612,Z 155,A 64.7027,B 20.3078,C -0.8525,E1 20.3873,E2 743.2199} C_DIS
LIN {X 54.2462,Y 119.6017,Z 155,A 62.7811,B 20.3077,C -0.8553,E1 20.3921,E2 745.1273} C_DIS
LIN {X 57.629,Y 118.0081,Z 155,A 61.1536,B 20.3077,C -0.8535,E1 20.3962,E2 746.7547} C_DIS
LIN {X 60.7624,Y 116.425,Z 155,A 59.5976,B 20.3079,C -0.8505,E1 20.4001,E2 748.3139} C_DIS
LIN {X 63.914,Y 114.7274,Z 155,A 57.5862,B 20.3087,C -0.8293,E1 20.4052,E2 750.3787} C_DIS
LIN {X 67.4945,Y 112.6581,Z 155,A 56.1485,B 20.3082,C -0.8421,E1 20.4085,E2 751.7741} C_DIS
LIN {X 71.247,Y 110.3233,Z 155,A 54.2694,B 20.3082,C -0.8412,E1 20.4129,E2 753.6482} C_DIS
LIN {X 74.7007,Y 108.0148,Z 155,A 52.5004,B 20.3082,C -0.8401,E1 20.417,E2 755.4129} C_DIS
LIN {X 78.0621,Y 105.6111,Z 155,A 50.605,B 20.3086,C -0.833,E1 20.4213,E2 757.3202} C_DIS
LIN {X 81.5572,Y 102.9357,Z 155,A 48.8712,B 20.3084,C -0.8375,E1 20.4251,E2 759.033} C_DIS
LIN {X 84.5383,Y 100.5016,Z 155,A 47.0928,B 20.3087,C -0.8301,E1 20.429,E2 760.8241} C_DIS
LIN {X 86.8595,Y 98.5024,Z 155,A 45.5749,B 20.3091,C -0.8197,E1 20.4322,E2 762.3644} C_DIS
LIN {X 91.2269,Y 94.472,Z 155,A 43.1479,B 20.3091,C -0.8215,E1 20.4371,E2 764.7736} C_DIS
LIN {X 94.5044,Y 91.1933,Z 155,A 41.155,B 20.3091,C -0.8184,E1 20.441,E2 766.7646} C_DIS
LIN {X 97.561,Y 87.9163,Z 155,A 39.1719,B 20.3093,C -0.8129,E1 20.4447,E2 768.7525} C_DIS
LIN {X 99.766,Y 85.4059,Z 155,A 37.6248,B 20.3096,C -0.8057,E1 20.4476,E2 770.3114} C_DIS
LIN {X 103.271,Y 81.1317,Z 155,A 35.3872,B 20.3096,C -0.8075,E1 20.4515,E2 772.5305} C_DIS
LIN {X 105.8276,Y 77.7675,Z 155,A 33.8317,B 20.3092,C -0.8156,E1 20.454,E2 774.0535} C_DIS
LIN {X 108.5955,Y 73.8536,Z 155,A 31.4165,B 20.31,C -0.7962,E1 20.458,E2 776.5094} C_DIS
LIN {X 111.1051,Y 70.0209,Z 155,A 29.4941,B 20.31,C -0.7945,E1 20.4608,E2 778.4248} C_DIS
LIN {X 113.1533,Y 66.6604,Z 155,A 27.7863,B 20.3102,C -0.7904,E1 20.4633,E2 780.1333} C_DIS
LIN {X 115.0983,Y 63.2441,Z 155,A 26.0104,B 20.3105,C -0.7831,E1 20.4657,E2 781.9184} C_DIS
LIN {X 116.65,Y 60.334,Z 155,A 24.6772,B 20.3105,C -0.7838,E1 20.4674,E2 783.2407} C_DIS
LIN {X 118.5198,Y 56.5668,Z 155,A 22.5545,B 20.3111,C -0.7661,E1 20.4701,E2 785.3997} C_DIS
LIN {X 119.973,Y 53.4162,Z 155,A 21.3686,B 20.3107,C -0.7763,E1 20.4714,E2 786.5484} C_DIS
LIN {X 121.333,Y 50.2516,Z 155,A 19.8566,B 20.3109,C -0.7716,E1 20.473,E2 788.0634} C_DIS
LIN {X 122.7299,Y 46.7404,Z 155,A 18.1619,B 20.3111,C -0.7648,E1 20.4748,E2 789.7657} C_DIS
LIN {X 124.0225,Y 43.1884,Z 155,A 16.6937,B 20.3111,C -0.768,E1 20.4761,E2 791.2144} C_DIS
LIN {X 125.0702,Y 40.053,Z 155,A 15.1514,B 20.3113,C -0.7593,E1 20.4775,E2 792.7706} C_DIS
LIN {X 125.9668,Y 37.138,Z 155,A 13.7843,B 20.3115,C -0.7537,E1 20.4786,E2 794.1439} C_DIS
LIN {X 126.8935,Y 33.8354,Z 155,A 11.9615,B 20.3122,C -0.7348,E1 20.4799,E2 796.0075} C_DIS
LIN {X 127.8559,Y 29.9978,Z 155,A 10.5618,B 20.3119,C -0.744,E1 20.4808,E2 797.3709} C_DIS
LIN {X 129.2391,Y 23.3267,Z 155,A 7.7101,B 20.3119,C -0.7402,E1 20.4824,E2 800.2123} C_DIS
LIN {X 129.7932,Y 20.0145,Z 155,A 6.2489,B 20.3121,C -0.7359,E1 20.483,E2 801.6752} C_DIS
LIN {X 130.5393,Y 14.3688,Z 155,A 3.5175,B 20.3128,C -0.7172,E1 20.4839,E2 804.4398} C_DIS
LIN {X 130.9897,Y 9.4123,Z 155,A 1.6246,B 20.3126,C -0.7228,E1 20.4844,E2 806.3027} C_DIS
LIN {X 131.1745,Y 6.3395,Z 155,A 0.2624,B 20.3128,C -0.7177,E1 20.4846,E2 807.6692} C_DIS
LIN {X 131.3092,Y 2.1919,Z 155,A -1.4793,B 20.3128,C -0.715,E1 20.4846,E2 809.4054} C_DIS
LIN {X 131.3123,Y -2.0061,Z 155,A -3.3064,B 20.313,C -0.7094,E1 20.4846,E2 811.2348} C_DIS
LIN {X 131.1982,Y -5.8682,Z 155,A -5.076,B 20.3133,C -0.7003,E1 20.4845,E2 813.0172} C_DIS
LIN {X 130.969,Y -9.6956,Z 155,A -6.4481,B 20.3131,C -0.7085,E1 20.4842,E2 814.3557} C_DIS
LIN {X 130.3494,Y -16.0029,Z 155,A -9.4708,B 20.3137,C -0.6882,E1 20.4834,E2 817.4139} C_DIS
LIN {X 129.6896,Y -20.6836,Z 155,A -11.8976,B 20.3145,C -0.6655,E1 20.4823,E2 819.8877} C_DIS
LIN {X 128.974,Y -24.7499,Z 155,A -13.1422,B 20.3139,C -0.6846,E1 20.4817,E2 821.0684} C_DIS
LIN {X 127.7963,Y -30.2523,Z 155,A -15.6939,B 20.3142,C -0.6726,E1 20.4802,E2 823.6359} C_DIS
LIN {X 126.7905,Y -34.2219,Z 155,A -18.2731,B 20.3155,C -0.632,E1 20.4782,E2 826.3127} C_DIS
LIN {X 125.0461,Y -40.1285,Z 155,A -20.1094,B 20.3146,C -0.6614,E1 20.4768,E2 828.0518} C_DIS
LIN {X 123.6739,Y -44.1779,Z 155,A -21.9311,B 20.3147,C -0.6577,E1 20.4751,E2 829.8713} C_DIS
LIN {X 120.44,Y -52.3548,Z 155,A -25.7716,B 20.3151,C -0.646,E1 20.4711,E2 833.7185} C_DIS
LIN {X 118.5149,Y -56.577,Z 155,A -28.475,B 20.3161,C -0.61,E1 20.4678,E2 836.5064} C_DIS
LIN {X 116.0198,Y -61.534,Z 155,A -30.1615,B 20.3154,C -0.6354,E1 20.4657,E2 838.109} C_DIS
LIN {X 113.9345,Y -65.3167,Z 155,A -32.1142,B 20.3156,C -0.627,E1 20.463,E2 840.0729} C_DIS
LIN {X 111.6838,Y -69.0949,Z 155,A -34.0316,B 20.3158,C -0.6217,E1 20.4602,E2 841.9932} C_DIS
LIN {X 109.3291,Y -72.7629,Z 155,A -35.8965,B 20.3159,C -0.6181,E1 20.4574,E2 843.8567} C_DIS
LIN {X 106.9179,Y -76.2617,Z 155,A -38.1285,B 20.3165,C -0.5965,E1 20.4537,E2 846.137} C_DIS
LIN {X 104.4671,Y -79.5845,Z 155,A -39.7432,B 20.3165,C -0.5999,E1 20.451,E2 847.7321} C_DIS
LIN {X 102.3999,Y -82.2289,Z 155,A -40.9503,B 20.3162,C -0.6075,E1 20.449,E2 848.9106} C_DIS
LIN {X 97.5217,Y -87.9598,Z 155,A -43.9772,B 20.3162,C -0.6105,E1 20.4435,E2 851.9114} C_DIS
LIN {X 92.9906,Y -92.7365,Z 155,A -47.0951,B 20.3166,C -0.5927,E1 20.4374,E2 855.0633} C_DIS
LIN {X 88.3591,Y -97.1594,Z 155,A -50.4319,B 20.3174,C -0.5626,E1 20.4305,E2 858.4692} C_DIS
LIN {X 84.5748,Y -100.4709,Z 155,A -51.9695,B 20.3168,C -0.5864,E1 20.4273,E2 859.9311} C_DIS
LIN {X 81.0992,Y -103.2963,Z 155,A -54.2946,B 20.3174,C -0.5661,E1 20.4222,E2 862.3035} C_DIS
LIN {X 78.14,Y -105.5534,Z 155,A -55.6704,B 20.3172,C -0.5736,E1 20.4191,E2 863.6518} C_DIS
LIN {X 74.3687,Y -108.2431,Z 155,A -57.5757,B 20.3172,C -0.5746,E1 20.4148,E2 865.5457} C_DIS
LIN {X 71.0029,Y -110.4804,Z 155,A -59.4085,B 20.3172,C -0.5683,E1 20.4105,E2 867.3891} C_DIS
LIN {X 67.1653,Y -112.8543,Z 155,A -61.2381,B 20.3172,C -0.5707,E1 20.4062,E2 869.2043} C_DIS
LIN {X 63.8319,Y -114.7729,Z 155,A -62.9953,B 20.3174,C -0.5644,E1 20.4019,E2 870.9732} C_DIS
LIN {X 56.9634,Y -118.3303,Z 155,A -66.3106,B 20.3174,C -0.5616,E1 20.3936,E2 874.2851} C_DIS
LIN {X 53.759,Y -119.8197,Z 155,A -67.8225,B 20.3175,C -0.5606,E1 20.3898,E2 875.7952} C_DIS
LIN {X 50.0383,Y -121.422,Z 155,A -69.9299,B 20.3179,C -0.5435,E1 20.3843,E2 877.9453} C_DIS
LIN {X 46.7499,Y -122.7263,Z 155,A -71.139,B 20.3176,C -0.5557,E1 20.3812,E2 879.1159} C_DIS
LIN {X 43.4614,Y -123.9278,Z 155,A -72.7161,B 20.3177,C -0.5517,E1 20.377,E2 880.7005} C_DIS
LIN {X 40.5706,Y -124.9049,Z 155,A -74.3941,B 20.3182,C -0.5354,E1 20.3725,E2 882.4213} C_DIS
LIN {X 36.9609,Y -126.0186,Z 155,A -76.0363,B 20.3182,C -0.5339,E1 20.3681,E2 884.0643} C_DIS
LIN {X 33.078,Y -127.0955,Z 155,A -77.5015,B 20.3179,C -0.5445,E1 20.3642,E2 885.4961} C_DIS
LIN {X 29.4277,Y -127.9877,Z 155,A -79.778,B 20.3186,C -0.5162,E1 20.3578,E2 887.85} C_DIS
LIN {X 23.7886,Y -129.1564,Z 155,A -81.5745,B 20.3179,C -0.5443,E1 20.3531,E2 889.5631} C_DIS
LIN {X 18.202,Y -130.0603,Z 155,A -84.1004,B 20.318,C -0.5403,E1 20.3461,E2 892.0976} C_DIS
LIN {X 13.2075,Y -130.6632,Z 155,A -86.2649,B 20.318,C -0.5403,E1 20.3401,E2 894.26} C_DIS
LIN {X 9.4789,Y -130.9849,Z 155,A -87.8085,B 20.318,C -0.5434,E1 20.3358,E2 895.7938} C_DIS
LIN {X 5.3341,Y -131.2192,Z 155,A -89.633,B 20.318,C -0.5422,E1 20.3307,E2 897.6209} C_DIS
LIN {X 1.4274,Y -131.3216,Z 155,A -91.3902,B 20.318,C -0.5395,E1 20.3258,E2 899.3854} C_DIS
LIN {X 1.4274,Y -131.3216,Z 155,A -91.3902,B 20.318,C -0.5395,E1 20.3258,E2 899.3854} C_DIS
Enddeposition()
LIN {X 0.9295,Y -130.3863,Z 155,A -91.0205,B 19.007,C -0.3878,E1 19.0117,E2 899.3461} C_DIS
Startdeposition()
$VEL.CP = VEL_PRINT
LIN {X 3.5164,Y -130.3448,Z 155,A -89.3214,B 19.0065,C -0.41,E1 19.0167,E2 897.5793} C_DIS
LIN {X 7.4127,Y -130.1826,Z 155,A -87.6077,B 19.0065,C -0.4106,E1 19.0215,E2 895.8646} C_DIS
LIN {X 10.84,Y -129.9408,Z 155,A -86.0846,B 19.0065,C -0.4118,E1 19.0257,E2 894.339} C_DIS
LIN {X 14.9616,Y -129.5317,Z 155,A -84.2387,B 19.0065,C -0.4137,E1 19.0308,E2 892.4888} C_DIS
LIN {X 17.9786,Y -129.1474,Z 155,A -82.2213,B 19.0058,C -0.4417,E1 19.0367,E2 890.3879} C_DIS
LIN {X 23.4071,Y -128.2745,Z 155,A -80.7386,B 19.0066,C -0.4061,E1 19.0404,E2 889.0165} C_DIS
LIN {X 29.2095,Y -127.0782,Z 155,A -77.8409,B 19.0063,C -0.42,E1 19.0485,E2 886.0814} C_DIS
LIN {X 32.7572,Y -126.2121,Z 155,A -75.9815,B 19.0061,C -0.4317,E1 19.0536,E2 884.1898} C_DIS
LIN {X 36.1713,Y -125.2753,Z 155,A -74.4718,B 19.0061,C -0.4315,E1 19.0576,E2 882.6844} C_DIS
LIN {X 39.3853,Y -124.3017,Z 155,A -73.1953,B 19.0061,C -0.4251,E1 19.0609,E2 881.4306} C_DIS
LIN {X 43.8994,Y -122.7801,Z 155,A -71.184,B 19.0062,C -0.4243,E1 19.0662,E2 879.4272} C_DIS
LIN {X 47.9251,Y -121.2671,Z 155,A -69.1962,B 19.0061,C -0.4307,E1 19.0714,E2 877.4258} C_DIS
LIN {X 52.5528,Y -119.3346,Z 155,A -67.043,B 19.0061,C -0.4317,E1 19.077,E2 875.2764} C_DIS
LIN {X 58.9074,Y -116.3269,Z 155,A -63.9292,B 19.0059,C -0.4374,E1 19.0848,E2 872.1563} C_DIS
LIN {X 63.3727,Y -113.9581,Z 155,A -61.8313,B 19.0059,C -0.4361,E1 19.0899,E2 870.0709} C_DIS
LIN {X 67.1243,Y -111.7899,Z 155,A -59.854,B 19.0059,C -0.4424,E1 19.0947,E2 868.0824} C_DIS
LIN {X 70.5848,Y -109.6375,Z 155,A -58.146,B 19.0059,C -0.4422,E1 19.0987,E2 866.3823} C_DIS
LIN {X 74.1297,Y -107.2727,Z 155,A -56.2109,B 19.0057,C -0.4484,E1 19.1032,E2 864.4372} C_DIS
LIN {X 77.6293,Y -104.7677,Z 155,A -53.6952,B 19.005,C -0.478,E1 19.109,E2 861.8431} C_DIS
LIN {X 82.0705,Y -101.3261,Z 155,A -51.91,B 19.0055,C -0.4548,E1 19.1127,E2 860.138} C_DIS
LIN {X 85.4491,Y -98.494,Z 155,A -49.9843,B 19.0055,C -0.4585,E1 19.1168,E2 858.2112} C_DIS
LIN {X 88.7412,Y -95.5379,Z 155,A -47.6165,B 19.0049,C -0.4805,E1 19.1218,E2 855.7892} C_DIS
LIN {X 91.9231,Y -92.4804,Z 155,A -46.161,B 19.0053,C -0.4648,E1 19.1246,E2 854.3898} C_DIS
LIN {X 94.4612,Y -89.8868,Z 155,A -44.4912,B 19.0051,C -0.4717,E1 19.1278,E2 852.7086} C_DIS
LIN {X 97.6219,Y -86.4433,Z 155,A -42.1347,B 19.0047,C -0.4894,E1 19.1323,E2 850.3125} C_DIS
LIN {X 100.2748,Y -83.3517,Z 155,A -40.7135,B 19.005,C -0.4784,E1 19.1348,E2 848.9335} C_DIS
LIN {X 103.3829,Y -79.4642,Z 155,A -37.9928,B 19.0043,C -0.5065,E1 19.1396,E2 846.1447} C_DIS
LIN {X 106.3805,Y -75.4039,Z 155,A -36.3231,B 19.0047,C -0.4893,E1 19.1422,E2 844.5385} C_DIS
LIN {X 108.8604,Y -71.7768,Z 155,A -34.4288,B 19.0047,C -0.4929,E1 19.1451,E2 842.6456} C_DIS
LIN {X 111.3043,Y -67.9259,Z 155,A -32.471,B 19.0045,C -0.4965,E1 19.148,E2 840.6905} C_DIS
LIN {X 113.4779,Y -64.2293,Z 155,A -30.6157,B 19.0045,C -0.5005,E1 19.1506,E2 838.8358} C_DIS
LIN {X 115.4629,Y -60.5829,Z 155,A -27.7792,B 19.0032,C -0.5486,E1 19.1544,E2 835.8729} C_DIS
LIN {X 118.6865,Y -54.0012,Z 155,A -25.6785,B 19.0042,C -0.5104,E1 19.1568,E2 833.904} C_DIS
LIN {X 121.7406,Y -46.707,Z 155,A -22.1365,B 19.0038,C -0.5234,E1 19.1605,E2 830.3487} C_DIS
LIN {X 123.1172,Y -42.9443,Z 155,A -20.4485,B 19.0038,C -0.5256,E1 19.1621,E2 828.6667} C_DIS
LIN {X 124.4148,Y -39.0311,Z 155,A -17.95,B 19.0028,C -0.5602,E1 19.1643,E2 826.0821} C_DIS
LIN {X 125.9073,Y -33.9039,Z 155,A -16.3202,B 19.0035,C -0.537,E1 19.1654,E2 824.5357} C_DIS
LIN {X 126.9503,Y -29.7694,Z 155,A -13.7843,B 19.0025,C -0.5708,E1 19.1671,E2 821.9166} C_DIS
LIN {X 128.0354,Y -24.6784,Z 155,A -12.4703,B 19.0035,C -0.5367,E1 19.1678,E2 820.7169} C_DIS
LIN {X 128.9901,Y -19.0797,Z 155,A -9.647,B 19.0029,C -0.5581,E1 19.1691,E2 817.8506} C_DIS
LIN {X 129.803,Y -12.3802,Z 155,A -6.7708,B 19.0027,C -0.5636,E1 19.17,E2 814.9806} C_DIS
LIN {X 130.1129,Y -8.5456,Z 155,A -5.0491,B 19.0025,C -0.5702,E1 19.1703,E2 813.2527} C_DIS
LIN {X 130.3032,Y -4.8226,Z 155,A -3.4015,B 19.0024,C -0.5757,E1 19.1705,E2 811.6015} C_DIS
LIN {X 130.3911,Y -0.6925,Z 155,A -1.7008,B 19.0024,C -0.5766,E1 19.1705,E2 809.9119} C_DIS
LIN {X 130.3518,Y 3.2645,Z 155,A -0.0565,B 19.0024,C -0.578,E1 19.1705,E2 808.2764} C_DIS
LIN {X 130.2745,Y 5.5534,Z 155,A 1.1137,B 19.002,C -0.588,E1 19.1704,E2 807.0851} C_DIS
LIN {X 130.0483,Y 9.4619,Z 155,A 2.5814,B 19.0022,C -0.5828,E1 19.1701,E2 805.6452} C_DIS
LIN {X 129.5499,Y 14.8095,Z 155,A 5.8778,B 19.0007,C -0.6296,E1 19.1691,E2 802.2325} C_DIS
LIN {X 128.7511,Y 20.6322,Z 155,A 7.6306,B 19.0016,C -0.6024,E1 19.1684,E2 800.5765} C_DIS
LIN {X 128.0106,Y 24.8083,Z 155,A 9.7303,B 19.0011,C -0.618,E1 19.1673,E2 798.4458} C_DIS
LIN {X 127.124,Y 29.0092,Z 155,A 11.84,B 19.0006,C -0.6331,E1 19.166,E2 796.3067} C_DIS
LIN {X 126.1057,Y 33.1599,Z 155,A 13.1447,B 19.0012,C -0.6145,E1 19.1651,E2 795.0687} C_DIS
LIN {X 125.3119,Y 36.0461,Z 155,A 14.7333,B 19.0007,C -0.6299,E1 19.1639,E2 793.4457} C_DIS
LIN {X 123.817,Y 40.8835,Z 155,A 16.7857,B 19.0007,C -0.6292,E1 19.1622,E2 791.4111} C_DIS
LIN {X 122.6229,Y 44.3356,Z 155,A 18.3606,B 19.0007,C -0.6325,E1 19.1607,E2 789.8379} C_DIS
LIN {X 121.2234,Y 48.0358,Z 155,A 20.1251,B 19.0004,C -0.6386,E1 19.1589,E2 788.0682} C_DIS
LIN {X 119.7185,Y 51.6669,Z 155,A 21.6901,B 19.0005,C -0.6367,E1 19.1572,E2 786.5206} C_DIS
LIN {X 118.4267,Y 54.5631,Z 155,A 23.6512,B 18.9996,C -0.6642,E1 19.1549,E2 784.4898} C_DIS
LIN {X 116.505,Y 58.5576,Z 155,A 25.0261,B 19.0002,C -0.6456,E1 19.1532,E2 783.1816} C_DIS
LIN {X 114.7395,Y 61.9467,Z 155,A 26.8308,B 18.9999,C -0.6553,E1 19.1508,E2 781.3601} C_DIS
LIN {X 112.6953,Y 65.5922,Z 155,A 28.6112,B 18.9999,C -0.6579,E1 19.1484,E2 779.5846} C_DIS
LIN {X 110.3961,Y 69.3919,Z 155,A 30.6096,B 18.9996,C -0.6648,E1 19.1454,E2 777.5786} C_DIS
LIN {X 108.7795,Y 71.8997,Z 155,A 32.2366,B 18.999,C -0.6812,E1 19.1429,E2 775.9126} C_DIS
LIN {X 106.5738,Y 75.1297,Z 155,A 33.7288,B 18.9992,C -0.6761,E1 19.1405,E2 774.4459} C_DIS
LIN {X 103.6815,Y 79.0737,Z 155,A 35.7473,B 18.9992,C -0.6759,E1 19.1372,E2 772.4412} C_DIS
LIN {X 101.9024,Y 81.3536,Z 155,A 37.2963,B 18.9987,C -0.6903,E1 19.1344,E2 770.8578} C_DIS
LIN {X 99.5418,Y 84.2259,Z 155,A 38.6055,B 18.999,C -0.6807,E1 19.1321,E2 769.586} C_DIS
LIN {X 96.8633,Y 87.2934,Z 155,A 40.3635,B 18.999,C -0.6834,E1 19.1289,E2 767.8304} C_DIS
LIN {X 93.9743,Y 90.3963,Z 155,A 42.2935,B 18.9987,C -0.6902,E1 19.1251,E2 765.8911} C_DIS
LIN {X 90.8468,Y 93.5381,Z 155,A 43.9512,B 18.999,C -0.6824,E1 19.1219,E2 764.2665} C_DIS
LIN {X 87.4297,Y 96.7398,Z 155,A 46.1923,B 18.9986,C -0.694,E1 19.1173,E2 762.0024} C_DIS
LIN {X 84.4411,Y 99.3588,Z 155,A 47.9201,B 18.9985,C -0.6966,E1 19.1136,E2 760.2758} C_DIS
LIN {X 81.1306,Y 102.0799,Z 155,A 49.8094,B 18.9983,C -0.7004,E1 19.1095,E2 758.3846} C_DIS
LIN {X 77.6731,Y 104.7351,Z 155,A 51.6953,B 18.9983,C -0.7025,E1 19.1053,E2 756.5014} C_DIS
LIN {X 74.3609,Y 107.1118,Z 155,A 53.4442,B 18.9983,C -0.7038,E1 19.1013,E2 754.7567} C_DIS
LIN {X 71.6664,Y 108.9331,Z 155,A 54.9539,B 18.998,C -0.7094,E1 19.0978,E2 753.2368} C_DIS
LIN {X 67.8344,Y 111.3604,Z 155,A 57.2593,B 18.9975,C -0.7249,E1 19.0922,E2 750.8938} C_DIS
LIN {X 64.6081,Y 113.262,Z 155,A 58.6634,B 18.9977,C -0.7176,E1 19.0889,E2 749.5178} C_DIS
LIN {X 60.5829,Y 115.4629,Z 155,A 60.4413,B 18.998,C -0.7109,E1 19.0846,E2 747.7673} C_DIS
LIN {X 57.1124,Y 117.2201,Z 155,A 62.1904,B 18.9978,C -0.7146,E1 19.0802,E2 746.0133} C_DIS
LIN {X 53.6836,Y 118.8288,Z 155,A 63.9419,B 18.9976,C -0.72,E1 19.0757,E2 744.2512} C_DIS
LIN {X 50.3859,Y 120.2633,Z 155,A 65.9189,B 18.997,C -0.7375,E1 19.0705,E2 742.227} C_DIS
LIN {X 46.4878,Y 121.8238,Z 155,A 67.4613,B 18.9974,C -0.7273,E1 19.0666,E2 740.7204} C_DIS
LIN {X 42.2906,Y 123.3438,Z 155,A 69.2378,B 18.9976,C -0.7218,E1 19.062,E2 738.9656} C_DIS
LIN {X 38.2881,Y 124.6437,Z 155,A 71.0108,B 18.9976,C -0.7203,E1 19.0573,E2 737.2017} C_DIS
LIN {X 34.3662,Y 125.7839,Z 155,A 73.019,B 18.9973,C -0.7299,E1 19.0518,E2 735.1686} C_DIS
LIN {X 30.7473,Y 126.7149,Z 155,A 74.4551,B 18.9975,C -0.7229,E1 19.048,E2 733.7567} C_DIS
LIN {X 27.3954,Y 127.4816,Z 155,A 76.0175,B 18.9975,C -0.7257,E1 19.0437,E2 732.1886} C_DIS
LIN {X 23.5135,Y 128.2555,Z 155,A 77.815,B 18.9973,C -0.7288,E1 19.0388,E2 730.3847} C_DIS
LIN {X 19.9819,Y 128.8518,Z 155,A 79.9935,B 18.9964,C -0.7529,E1 19.0326,E2 728.1351} C_DIS
LIN {X 14.8608,Y 129.5437,Z 155,A 81.6641,B 18.9973,C -0.7301,E1 19.0281,E2 726.5362} C_DIS
LIN {X 10.3991,Y 129.978,Z 155,A 83.6592,B 18.9973,C -0.7313,E1 19.0226,E2 724.5388} C_DIS
LIN {X 6.5069,Y 130.2297,Z 155,A 85.5636,B 18.9969,C -0.7387,E1 19.0172,E2 722.6127} C_DIS
LIN {X 1.0236,Y 130.3885,Z 155,A 87.7584,B 18.9973,C -0.7302,E1 19.0112,E2 720.4444} C_DIS
LIN {X -3.2526,Y 130.3521,Z 155,A 89.634,B 18.9973,C -0.7298,E1 19.0059,E2 718.5701} C_DIS
LIN {X -7.3355,Y 130.1874,Z 155,A 91.301,B 18.9975,C -0.7244,E1 19.0013,E2 716.9192} C_DIS
LIN {X -10.1296,Y 129.9993,Z 155,A 93.1086,B 18.9967,C -0.7458,E1 18.9961,E2 715.0446} C_DIS
LIN {X -14.36,Y 129.5995,Z 155,A 94.2103,B 18.9978,C -0.716,E1 18.9933,E2 714.0337} C_DIS
LIN {X -19.6381,Y 128.905,Z 155,A 96.8449,B 18.9974,C -0.7257,E1 18.9859,E2 711.3664} C_DIS
LIN {X -27.0409,Y 127.5581,Z 155,A 100.0237,B 18.9977,C -0.7186,E1 18.9773,E2 708.2052} C_DIS
LIN {X -32.7309,Y 126.2187,Z 155,A 102.6769,B 18.9977,C -0.7195,E1 18.97,E2 705.5443} C_DIS
LIN {X -35.8645,Y 125.3649,Z 155,A 104.1075,B 18.9977,C -0.7182,E1 18.9662,E2 704.1145} C_DIS
LIN {X -38.8583,Y 124.4692,Z 155,A 105.7431,B 18.9974,C -0.7265,E1 18.9617,E2 702.4495} C_DIS
LIN {X -43.3518,Y 122.976,Z 155,A 107.7287,B 18.9976,C -0.7206,E1 18.9565,E2 700.477} C_DIS
LIN {X -46.6379,Y 121.7675,Z 155,A 109.0598,B 18.998,C -0.7111,E1 18.9531,E2 699.1715} C_DIS
LIN {X -52.5946,Y 119.3158,Z 155,A 112.0851,B 18.9978,C -0.7144,E1 18.9453,E2 696.1265} C_DIS
LIN {X -56.5041,Y 117.5133,Z 155,A 113.9104,B 18.998,C -0.7093,E1 18.9407,E2 694.3109} C_DIS
LIN {X -60.448,Y 115.5337,Z 155,A 115.7059,B 18.9983,C -0.7011,E1 18.9363,E2 692.5343} C_DIS
LIN {X -63.8373,Y 113.6982,Z 155,A 117.6227,B 18.9981,C -0.7064,E1 18.9315,E2 690.5934} C_DIS
LIN {X -67.7347,Y 111.4207,Z 155,A 119.5893,B 18.9983,C -0.7024,E1 18.9268,E2 688.6312} C_DIS
LIN {X -71.2624,Y 109.1982,Z 155,A 121.469,B 18.9983,C -0.7008,E1 18.9224,E2 686.7481} C_DIS
LIN {X -74.9202,Y 106.7217,Z 155,A 123.3976,B 18.9985,C -0.6967,E1 18.918,E2 684.8234} C_DIS
LIN {X -78.3379,Y 104.2388,Z 155,A 125.2974,B 18.9985,C -0.6947,E1 18.9137,E2 682.9208} C_DIS
LIN {X -81.9929,Y 101.3887,Z 155,A 127.3168,B 18.9987,C -0.6899,E1 18.9093,E2 680.906} C_DIS
LIN {X -85.3369,Y 98.591,Z 155,A 129.2454,B 18.9988,C -0.6863,E1 18.9052,E2 678.9785} C_DIS
LIN {X -88.4818,Y 95.7787,Z 155,A 131.0888,B 18.999,C -0.6818,E1 18.9014,E2 677.1388} C_DIS
LIN {X -91.5792,Y 92.8218,Z 155,A 133.0104,B 18.999,C -0.679,E1 18.8975,E2 675.2151} C_DIS
LIN {X -94.5115,Y 89.8342,Z 155,A 134.8315,B 18.9993,C -0.674,E1 18.894,E2 673.3987} C_DIS
LIN {X -97.3878,Y 86.7078,Z 155,A 136.7715,B 18.9993,C -0.6722,E1 18.8904,E2 671.4528} C_DIS
LIN {X -100.2928,Y 83.3299,Z 155,A 138.7238,B 18.9995,C -0.6671,E1 18.8869,E2 669.504} C_DIS
LIN {X -103.1062,Y 79.8223,Z 155,A 140.6902,B 18.9997,C -0.6618,E1 18.8835,E2 667.5415} C_DIS
LIN {X -105.82,Y 76.1891,Z 155,A 142.7399,B 18.9997,C -0.6586,E1 18.8801,E2 665.4881} C_DIS
LIN {X -108.3524,Y 72.5414,Z 155,A 144.6715,B 19,C -0.6528,E1 18.877,E2 663.5617} C_DIS
LIN {X -110.4344,Y 69.3312,Z 155,A 146.2826,B 19.0002,C -0.6457,E1 18.8746,E2 661.9612} C_DIS
LIN {X -112.7525,Y 65.4934,Z 155,A 148.3277,B 19.0003,C -0.643,E1 18.8717,E2 659.9103} C_DIS
LIN {X -114.8054,Y 61.8242,Z 155,A 150.3568,B 19.0003,C -0.6442,E1 18.869,E2 657.8629} C_DIS
LIN {X -117.2101,Y 57.1313,Z 155,A 152.8078,B 19.0003,C -0.6424,E1 18.8659,E2 655.3997} C_DIS
LIN {X -118.7321,Y 53.8998,Z 155,A 154.1816,B 19.0007,C -0.6309,E1 18.8644,E2 654.0513} C_DIS
LIN {X -120.3059,Y 50.2839,Z 155,A 155.6462,B 19.0011,C -0.6164,E1 18.8628,E2 652.6205} C_DIS
LIN {X -121.4725,Y 47.3966,Z 155,A 157.1334,B 19.0011,C -0.6166,E1 18.8612,E2 651.1216} C_DIS
LIN {X -122.6481,Y 44.2655,Z 155,A 158.6267,B 19.0013,C -0.613,E1 18.8598,E2 649.6278} C_DIS
LIN {X -123.714,Y 41.1927,Z 155,A 160.0359,B 19.0014,C -0.608,E1 18.8585,E2 648.2231} C_DIS
LIN {X -124.6628,Y 38.2258,Z 155,A 161.4551,B 19.0014,C -0.6057,E1 18.8573,E2 646.8002} C_DIS
LIN {X -125.4367,Y 35.6079,Z 155,A 162.7209,B 19.0015,C -0.6044,E1 18.8564,E2 645.5285} C_DIS
LIN {X -126.2774,Y 32.4999,Z 155,A 164.1302,B 19.0017,C -0.5999,E1 18.8554,E2 644.122} C_DIS
LIN {X -127.1098,Y 29.0714,Z 155,A 165.6131,B 19.0019,C -0.5927,E1 18.8544,E2 642.6494} C_DIS
LIN {X -127.9383,Y 25.1862,Z 155,A 167.6818,B 19.0017,C -0.5987,E1 18.8533,E2 640.5456} C_DIS
LIN {X -128.7609,Y 20.569,Z 155,A 169.5394,B 19.0021,C -0.5852,E1 18.8524,E2 638.715} C_DIS
LIN {X -129.2669,Y 17.0926,Z 155,A 171.0684,B 19.0023,C -0.5799,E1 18.8518,E2 637.19} C_DIS
LIN {X -129.666,Y 13.7423,Z 155,A 172.7351,B 19.0023,C -0.5818,E1 18.8513,E2 635.5039} C_DIS
LIN {X -130.2202,Y 6.6952,Z 155,A 175.6427,B 19.0027,C -0.5651,E1 18.8507,E2 632.6243} C_DIS
LIN {X -130.3934,Y 0.2916,Z 155,A 178.5984,B 19.0027,C -0.5612,E1 18.8506,E2 629.6564} C_DIS
LIN {X -130.2237,Y -6.6264,Z 155,A -178.3851,B 19.0031,C -0.5509,E1 18.8509,E2 626.6472} C_DIS
LIN {X -129.9216,Y -11.0671,Z 155,A -175.9899,B 19.0028,C -0.5604,E1 18.8514,E2 624.2031} C_DIS
LIN {X -129.5257,Y -15.0116,Z 155,A -174.4108,B 19.0031,C -0.5492,E1 18.8519,E2 622.6456} C_DIS
LIN {X -128.8825,Y -19.7835,Z 155,A -172.5372,B 19.0035,C -0.5342,E1 18.8526,E2 620.8034} C_DIS
LIN {X -128.3197,Y -23.1546,Z 155,A -171.0338,B 19.0037,C -0.5297,E1 18.8533,E2 619.3019} C_DIS
LIN {X -127.5478,Y -27.0886,Z 155,A -169.1858,B 19.0037,C -0.5274,E1 18.8544,E2 617.4461} C_DIS
LIN {X -126.761,Y -30.5563,Z 155,A -167.61,B 19.0038,C -0.5232,E1 18.8554,E2 615.8708} C_DIS
LIN {X -125.7542,Y -34.4724,Z 155,A -165.7944,B 19.0039,C -0.5193,E1 18.8567,E2 614.053} C_DIS
LIN {X -124.6809,Y -38.1666,Z 155,A -164.1786,B 19.0041,C -0.5117,E1 18.858,E2 612.448} C_DIS
LIN {X -123.4586,Y -41.9595,Z 155,A -161.6373,B 19.0035,C -0.5349,E1 18.8603,E2 609.8154} C_DIS
LIN {X -121.5769,Y -47.1282,Z 155,A -159.9818,B 19.0044,C -0.5007,E1 18.8619,E2 608.253} C_DIS
LIN {X -120.2665,Y -50.3783,Z 155,A -158.4072,B 19.0045,C -0.4976,E1 18.8635,E2 606.6761} C_DIS
LIN {X -119.0612,Y -53.164,Z 155,A -156.7759,B 19.0043,C -0.5045,E1 18.8654,E2 605.0112} C_DIS
LIN {X -117.7049,Y -56.103,Z 155,A -155.6625,B 19.0047,C -0.4896,E1 18.8667,E2 603.936} C_DIS
LIN {X -116.2637,Y -59.0317,Z 155,A -154.2739,B 19.0048,C -0.4841,E1 18.8684,E2 602.5542} C_DIS
LIN {X -114.4576,Y -62.4655,Z 155,A -151.8772,B 19.0043,C -0.5044,E1 18.8717,E2 600.0774} C_DIS
LIN {X -112.0941,Y -66.614,Z 155,A -150.3351,B 19.005,C -0.4789,E1 18.8738,E2 598.6035} C_DIS
LIN {X -110.0956,Y -69.868,Z 155,A -148.2756,B 19.0047,C -0.4884,E1 18.877,E2 596.5004} C_DIS
LIN {X -108.0533,Y -72.9862,Z 155,A -146.9389,B 19.0051,C -0.4734,E1 18.879,E2 595.201} C_DIS
LIN {X -105.4993,Y -76.6316,Z 155,A -144.9652,B 19.0051,C -0.4693,E1 18.8822,E2 593.227} C_DIS
LIN {X -102.8916,Y -80.0992,Z 155,A -143.2997,B 19.0055,C -0.456,E1 18.8849,E2 591.5917} C_DIS
LIN {X -101.0315,Y -82.4325,Z 155,A -141.7602,B 19.0054,C -0.4613,E1 18.8877,E2 590.0263} C_DIS
LIN {X -98.4861,Y -85.4581,Z 155,A -139.9678,B 19.0054,C -0.4593,E1 18.891,E2 588.2288} C_DIS
LIN {X -96.1443,Y -88.0841,Z 155,A -138.4129,B 19.0055,C -0.4563,E1 18.8939,E2 586.674} C_DIS
LIN {X -93.1081,Y -91.2873,Z 155,A -136.5024,B 19.0056,C -0.4511,E1 18.8976,E2 584.7683} C_DIS
LIN {X -90.1559,Y -94.204,Z 155,A -134.6388,B 19.0056,C -0.4488,E1 18.9013,E2 582.9011} C_DIS
LIN {X -86.8782,Y -97.2352,Z 155,A -132.6559,B 19.0057,C -0.4458,E1 18.9054,E2 580.9169} C_DIS
LIN {X -83.6031,Y -100.0654,Z 155,A -130.7913,B 19.0059,C -0.4408,E1 18.9094,E2 579.0579} C_DIS
LIN {X -80.2683,Y -102.7599,Z 155,A -128.8427,B 19.0059,C -0.4398,E1 18.9136,E2 577.1026} C_DIS
LIN {X -77.1242,Y -105.1396,Z 155,A -127.1814,B 19.006,C -0.4342,E1 18.9173,E2 575.4506} C_DIS
LIN {X -73.999,Y -107.362,Z 155,A -125.4104,B 19.006,C -0.4346,E1 18.9214,E2 573.6701} C_DIS
LIN {X -71.2198,Y -109.2258,Z 155,A -123.7851,B 19.006,C -0.4381,E1 18.9253,E2 572.0268} C_DIS
LIN {X -65.6106,Y -112.6847,Z 155,A -121.0124,B 19.0061,C -0.4293,E1 18.9319,E2 569.2699} C_DIS
LIN {X -62.2595,Y -114.57,Z 155,A -119.2629,B 19.0061,C -0.4293,E1 18.9361,E2 567.5137} C_DIS
LIN {X -58.3581,Y -116.6056,Z 155,A -117.2706,B 19.0061,C -0.4291,E1 18.9411,E2 565.5147} C_DIS
LIN {X -53.9167,Y -118.7246,Z 155,A -115.3767,B 19.0064,C -0.4164,E1 18.9458,E2 563.6534} C_DIS
LIN {X -49.8124,Y -120.5023,Z 155,A -113.1204,B 19.0062,C -0.4254,E1 18.9517,E2 561.3625} C_DIS
LIN {X -45.5776,Y -122.1667,Z 155,A -111.4426,B 19.0065,C -0.4113,E1 18.956,E2 559.7232} C_DIS
LIN {X -42.8481,Y -123.1506,Z 155,A -110.018,B 19.0064,C -0.4159,E1 18.9598,E2 558.2808} C_DIS
LIN {X -39.9247,Y -124.1294,Z 155,A -108.5394,B 19.0064,C -0.4195,E1 18.9638,E2 556.7873} C_DIS
LIN {X -35.3095,Y -125.5201,Z 155,A -106.5207,B 19.0064,C -0.4143,E1 18.9691,E2 554.7805} C_DIS
LIN {X -31.3502,Y -126.5692,Z 155,A -104.8041,B 19.0065,C -0.41,E1 18.9738,E2 553.0737} C_DIS
LIN {X -28.7128,Y -127.1917,Z 155,A -103.4628,B 19.0065,C -0.4152,E1 18.9775,E2 551.714} C_DIS
LIN {X -24.4876,Y -128.0719,Z 155,A -101.7089,B 19.0065,C -0.4089,E1 18.9822,E2 549.9769} C_DIS
LIN {X -17.8142,Y -129.1695,Z 155,A -98.8118,B 19.0066,C -0.405,E1 18.9902,E2 547.0881} C_DIS
LIN {X -14.033,Y -129.6347,Z 155,A -97.0421,B 19.0066,C -0.4084,E1 18.9951,E2 545.3064} C_DIS
LIN {X -10.1846,Y -129.9956,Z 155,A -95.2613,B 19.0065,C -0.4115,E1 19.0001,E2 543.5152} C_DIS
LIN {X -6.6793,Y -130.221,Z 155,A -93.7755,B 19.0065,C -0.4093,E1 19.0042,E2 542.0355} C_DIS
LIN {X -2.4152,Y -130.37,Z 155,A -91.9129,B 19.0065,C -0.409,E1 19.0094,E2 540.1736} C_DIS
LIN {X 0.9295,Y -130.3863,Z 155,A -91.0175,B 19.007,C -0.3869,E1 19.0118,E2 539.3461} C_DIS
Enddeposition()
LIN {X 0.9295,Y -130.3863,Z 155,A -91.0175,B 19.007,C -0.3869,E1 19.0118,E2 539.3461} C_DIS
Startdeposition()
$VEL.CP = VEL_PRINT
LIN {X -1.5566,Y -129.4489,Z 155,A -91.4278,B 16.1508,C -0.0834,E1 16.1485,E2 540.5561} C_DIS
LIN {X -5.7666,Y -129.3304,Z 155,A -93.2059,B 16.1508,C -0.0861,E1 16.1436,E2 542.325} C_DIS
LIN {X -9.3049,Y -129.122,Z 155,A -94.8072,B 16.1508,C -0.0851,E1 16.1391,E2 543.9307} C_DIS
LIN {X -13.0114,Y -128.8029,Z 155,A -96.8717,B 16.1509,C -0.0719,E1 16.1332,E2 546.0446} C_DIS
LIN {X -16.6939,Y -128.3759,Z 155,A -99.0131,B 16.1509,C -0.0564,E1 16.1272,E2 548.2444} C_DIS
LIN {X -22.949,Y -127.4064,Z 155,A -101.2433,B 16.1509,C -0.0755,E1 16.1212,E2 550.4092} C_DIS
LIN {X -26.4251,Y -126.7325,Z 155,A -102.4002,B 16.1509,C -0.0892,E1 16.1182,E2 551.5187} C_DIS
LIN {X -30.4076,Y -125.8348,Z 155,A -104.3277,B 16.1509,C -0.0864,E1 16.1129,E2 553.4606} C_DIS
LIN {X -33.684,Y -124.998,Z 155,A -105.7828,B 16.1509,C -0.0886,E1 16.109,E2 554.9111} C_DIS
LIN {X -37.013,Y -124.0543,Z 155,A -107.4902,B 16.1509,C -0.0841,E1 16.1043,E2 556.6392} C_DIS
LIN {X -41.6573,Y -122.5735,Z 155,A -109.4516,B 16.1509,C -0.092,E1 16.0992,E2 558.5779} C_DIS
LIN {X -45.9559,Y -121.0263,Z 155,A -112.0397,B 16.1509,C -0.0761,E1 16.0923,E2 561.2317} C_DIS
LIN {X -49.966,Y -119.4251,Z 155,A -113.847,B 16.1509,C -0.0813,E1 16.0876,E2 563.0269} C_DIS
LIN {X -53.6261,Y -117.8295,Z 155,A -115.4602,B 16.1509,C -0.088,E1 16.0836,E2 564.6222} C_DIS
LIN {X -57.4419,Y -116.0147,Z 155,A -117.1668,B 16.1508,C -0.0953,E1 16.0793,E2 566.3095} C_DIS
LIN {X -61.3779,Y -113.9834,Z 155,A -118.9558,B 16.1508,C -0.1031,E1 16.0749,E2 568.0784} C_DIS
LIN {X -64.3289,Y -112.3445,Z 155,A -121.2962,B 16.1508,C -0.0792,E1 16.0691,E2 570.5163} C_DIS
LIN {X -69.0318,Y -109.5174,Z 155,A -122.7999,B 16.1507,C -0.111,E1 16.0657,E2 571.9124} C_DIS
LIN {X -71.496,Y -107.9254,Z 155,A -124.588,B 16.1507,C -0.098,E1 16.0614,E2 573.757} C_DIS
LIN {X -74.9276,Y -105.5719,Z 155,A -126.2573,B 16.1507,C -0.1062,E1 16.0577,E2 575.4058} C_DIS
LIN {X -78.5106,Y -102.9347,Z 155,A -128.2059,B 16.1507,C -0.1102,E1 16.0533,E2 577.3513} C_DIS
LIN {X -81.8516,Y -100.2984,Z 155,A -130.0534,B 16.1507,C -0.1146,E1 16.0493,E2 579.1938} C_DIS
LIN {X -84.9353,Y -97.701,Z 155,A -131.8379,B 16.1507,C -0.1179,E1 16.0455,E2 580.9775} C_DIS
LIN {X -87.9497,Y -94.997,Z 155,A -133.7363,B 16.1507,C -0.1182,E1 16.0416,E2 582.8872} C_DIS
LIN {X -91.3378,Y -91.7435,Z 155,A -135.7716,B 16.1506,C -0.1237,E1 16.0375,E2 584.9163} C_DIS
LIN {X -94.3652,Y -88.627,Z 155,A -137.667,B 16.1506,C -0.1285,E1 16.0338,E2 586.8073} C_DIS
LIN {X -96.9306,Y -85.8132,Z 155,A -139.3896,B 16.1506,C -0.1311,E1 16.0306,E2 588.5332} C_DIS
LIN {X -99.4813,Y -82.8435,Z 155,A -141.5382,B 16.1506,C -0.1226,E1 16.0267,E2 590.7285} C_DIS
LIN {X -101.9807,Y -79.7463,Z 155,A -142.9259,B 16.1505,C -0.1377,E1 16.0244,E2 592.072} C_DIS
LIN {X -104.1061,Y -76.9513,Z 155,A -144.5515,B 16.1505,C -0.1392,E1 16.0216,E2 593.7047} C_DIS
LIN {X -106.726,Y -73.2735,Z 155,A -146.5816,B 16.1505,C -0.1431,E1 16.0184,E2 595.7369} C_DIS
LIN {X -109.1434,Y -69.622,Z 155,A -148.4639,B 16.1504,C -0.1495,E1 16.0155,E2 597.6112} C_DIS
LIN {X -111.3617,Y -66.016,Z 155,A -150.2668,B 16.1504,C -0.1563,E1 16.0129,E2 599.4043} C_DIS
LIN {X -113.5273,Y -62.2179,Z 155,A -152.1178,B 16.1502,C -0.1638,E1 16.0104,E2 601.2439} C_DIS
LIN {X -114.8484,Y -59.7414,Z 155,A -153.4435,B 16.1502,C -0.1646,E1 16.0087,E2 602.578} C_DIS
LIN {X -116.292,Y -56.8797,Z 155,A -155.0353,B 16.1502,C -0.1633,E1 16.0067,E2 604.1884} C_DIS
LIN {X -117.7385,Y -53.8229,Z 155,A -156.3546,B 16.1502,C -0.1725,E1 16.0051,E2 605.4859} C_DIS
LIN {X -119.0545,Y -50.8459,Z 155,A -157.815,B 16.1502,C -0.1758,E1 16.0035,E2 606.9472} C_DIS
LIN {X -120.3078,Y -47.8059,Z 155,A -159.2922,B 16.1501,C -0.1792,E1 16.002,E2 608.4255} C_DIS
LIN {X -121.457,Y -44.8061,Z 155,A -160.7185,B 16.1501,C -0.1831,E1 16.0006,E2 609.8508} C_DIS
LIN {X -122.849,Y -40.8301,Z 155,A -162.648,B 16.1501,C -0.1864,E1 15.9988,E2 611.7858} C_DIS
LIN {X -123.895,Y -37.5384,Z 155,A -164.196,B 16.15,C -0.1902,E1 15.9975,E2 613.3344} C_DIS
LIN {X -124.8347,Y -34.2877,Z 155,A -165.6508,B 16.15,C -0.1958,E1 15.9964,E2 614.7825} C_DIS
LIN {X -125.5217,Y -31.6756,Z 155,A -166.9745,B 16.15,C -0.1956,E1 15.9955,E2 616.1196} C_DIS
LIN {X -126.3066,Y -28.3876,Z 155,A -168.4433,B 16.1498,C -0.2007,E1 15.9946,E2 617.5835} C_DIS
LIN {X -126.9493,Y -25.3595,Z 155,A -169.7571,B 16.1498,C -0.2064,E1 15.9938,E2 618.8893} C_DIS
LIN {X -127.5733,Y -22.0134,Z 155,A -171.2832,B 16.1498,C -0.2103,E1 15.9931,E2 620.4159} C_DIS
LIN {X -127.9994,Y -19.375,Z 155,A -172.4622,B 16.1497,C -0.2139,E1 15.9926,E2 621.5931} C_DIS
LIN {X -128.3517,Y -16.8788,Z 155,A -173.621,B 16.1497,C -0.216,E1 15.9921,E2 622.7554} C_DIS
LIN {X -128.7694,Y -13.3329,Z 155,A -175.1632,B 16.1496,C -0.2219,E1 15.9916,E2 624.2914} C_DIS
LIN {X -129.0572,Y -10.188,Z 155,A -176.6159,B 16.1496,C -0.2245,E1 15.9913,E2 625.7486} C_DIS
LIN {X -129.3312,Y -5.7459,Z 155,A -178.8202,B 16.1496,C -0.2237,E1 15.991,E2 627.9772} C_DIS
LIN {X -129.4339,Y -2.4621,Z 155,A 179.8467,B 16.1494,C -0.2316,E1 15.9909,E2 629.2946} C_DIS
LIN {X -129.4464,Y 1.7062,Z 155,A 177.8678,B 16.1494,C -0.2334,E1 15.9909,E2 631.2865} C_DIS
LIN {X -129.3127,Y 6.1199,Z 155,A 176.0615,B 16.1493,C -0.2435,E1 15.9911,E2 633.0734} C_DIS
LIN {X -129.0469,Y 10.3107,Z 155,A 174.222,B 16.1492,C -0.2497,E1 15.9914,E2 634.9083} C_DIS
LIN {X -128.8139,Y 12.8958,Z 155,A 172.8555,B 16.1492,C -0.247,E1 15.9918,E2 636.298} C_DIS
LIN {X -128.2638,Y 17.5491,Z 155,A 170.9489,B 16.1491,C -0.258,E1 15.9925,E2 638.1828} C_DIS
LIN {X -127.8932,Y 20.0605,Z 155,A 169.6539,B 16.1491,C -0.2565,E1 15.993,E2 639.4958} C_DIS
LIN {X -127.2816,Y 23.6382,Z 155,A 168.2068,B 16.1489,C -0.2659,E1 15.9937,E2 640.9226} C_DIS
LIN {X -126.8036,Y 26.0756,Z 155,A 167.0567,B 16.1489,C -0.2678,E1 15.9944,E2 642.077} C_DIS
LIN {X -125.9779,Y 29.8139,Z 155,A 165.3409,B 16.1489,C -0.2722,E1 15.9954,E2 643.7929} C_DIS
LIN {X -125.2423,Y 32.7679,Z 155,A 164.0677,B 16.1487,C -0.2784,E1 15.9963,E2 645.0559} C_DIS
LIN {X -124.6034,Y 35.1147,Z 155,A 162.923,B 16.1487,C -0.2796,E1 15.9972,E2 646.2068} C_DIS
LIN {X -123.8152,Y 37.7993,Z 155,A 161.5548,B 16.1487,C -0.2796,E1 15.9983,E2 647.588} C_DIS
LIN {X -122.7179,Y 41.2239,Z 155,A 159.9422,B 16.1487,C -0.2836,E1 15.9997,E2 649.2008} C_DIS
LIN {X -121.3111,Y 45.1955,Z 155,A 158.081,B 16.1485,C -0.2891,E1 16.0014,E2 651.059} C_DIS
LIN {X -119.9327,Y 48.7363,Z 155,A 156.4668,B 16.1485,C -0.2958,E1 16.0031,E2 652.6634} C_DIS
LIN {X -118.8095,Y 51.4127,Z 155,A 155.0481,B 16.1485,C -0.2956,E1 16.0047,E2 654.0954} C_DIS
LIN {X -116.2053,Y 57.0555,Z 155,A 152.2868,B 16.1483,C -0.303,E1 16.008,E2 656.8542} C_DIS
LIN {X -112.8469,Y 63.4432,Z 155,A 149.3518,B 16.148,C -0.3192,E1 16.0118,E2 659.7556} C_DIS
LIN {X -109.926,Y 68.3792,Z 155,A 146.6034,B 16.148,C -0.3199,E1 16.0157,E2 662.5245} C_DIS
LIN {X -107.859,Y 71.596,Z 155,A 144.8745,B 16.148,C -0.3232,E1 16.0184,E2 664.2554} C_DIS
LIN {X -105.5601,Y 74.9445,Z 155,A 142.9398,B 16.1479,C -0.3238,E1 16.0215,E2 666.2032} C_DIS
LIN {X -102.8742,Y 78.5897,Z 155,A 140.9745,B 16.1478,C -0.33,E1 16.0248,E2 668.1614} C_DIS
LIN {X -100.1669,Y 82.0125,Z 155,A 139.0535,B 16.1477,C -0.335,E1 16.0281,E2 670.0788} C_DIS
LIN {X -97.3634,Y 85.3222,Z 155,A 137.0731,B 16.1477,C -0.3378,E1 16.0317,E2 672.0636} C_DIS
LIN {X -94.4192,Y 88.5697,Z 155,A 135.0836,B 16.1476,C -0.3408,E1 16.0355,E2 674.0562} C_DIS
LIN {X -91.2662,Y 91.8146,Z 155,A 133.1102,B 16.1474,C -0.3462,E1 16.0394,E2 676.0237} C_DIS
LIN {X -88.0219,Y 94.9298,Z 155,A 131.0922,B 16.1474,C -0.3497,E1 16.0435,E2 678.0424} C_DIS
LIN {X -84.7549,Y 97.858,Z 155,A 129.1167,B 16.1474,C -0.3527,E1 16.0476,E2 680.0194} C_DIS
LIN {X -81.3623,Y 100.6957,Z 155,A 127.1933,B 16.1472,C -0.3577,E1 16.0517,E2 681.9366} C_DIS
LIN {X -78.0098,Y 103.3146,Z 155,A 125.2855,B 16.1472,C -0.3606,E1 16.056,E2 683.845} C_DIS
LIN {X -74.7695,Y 105.6835,Z 155,A 123.5813,B 16.147,C -0.3661,E1 16.0598,E2 685.539} C_DIS
LIN {X -71.8949,Y 107.6595,Z 155,A 121.9441,B 16.147,C -0.3661,E1 16.0636,E2 687.185} C_DIS
LIN {X -68.0974,Y 110.1014,Z 155,A 120.0435,B 16.1469,C -0.3724,E1 16.0681,E2 689.0724} C_DIS
LIN {X -64.8847,Y 112.0242,Z 155,A 118.2431,B 16.1469,C -0.3708,E1 16.0724,E2 690.8873} C_DIS
LIN {X -61.7421,Y 113.7868,Z 155,A 116.5851,B 16.1469,C -0.3714,E1 16.0765,E2 692.5508} C_DIS
LIN {X -58.47,Y 115.5001,Z 155,A 115.053,B 16.1468,C -0.3769,E1 16.0803,E2 694.0696} C_DIS
LIN {X -54.3224,Y 117.5076,Z 155,A 112.9943,B 16.1468,C -0.3792,E1 16.0855,E2 696.1284} C_DIS
LIN {X -50.2609,Y 119.302,Z 155,A 110.9124,B 16.1468,C -0.3782,E1 16.0908,E2 698.2217} C_DIS
LIN {X -46.7712,Y 120.7122,Z 155,A 109.4047,B 16.1466,C -0.3851,E1 16.0947,E2 699.71} C_DIS
LIN {X -42.8837,Y 122.1483,Z 155,A 107.3759,B 16.1466,C -0.3812,E1 16.1001,E2 701.7592} C_DIS
LIN {X -38.8226,Y 123.4996,Z 155,A 105.7277,B 16.1465,C -0.3907,E1 16.1044,E2 703.3779} C_DIS
LIN {X -35.4346,Y 124.514,Z 155,A 104.2092,B 16.1464,C -0.3936,E1 16.1084,E2 704.8898} C_DIS
LIN {X -32.6977,Y 125.261,Z 155,A 102.5833,B 16.1466,C -0.3833,E1 16.1129,E2 706.5567} C_DIS
LIN {X -28.795,Y 126.2135,Z 155,A 101.0328,B 16.1464,C -0.3918,E1 16.1171,E2 708.0801} C_DIS
LIN {X -22.9082,Y 127.4137,Z 155,A 98.5019,B 16.1463,C -0.3976,E1 16.124,E2 710.5946} C_DIS
LIN {X -19.5631,Y 127.9702,Z 155,A 96.8706,B 16.1463,C -0.3944,E1 16.1285,E2 712.2397} C_DIS
LIN {X -15.866,Y 128.4819,Z 155,A 95.0618,B 16.1465,C -0.3903,E1 16.1335,E2 714.0653} C_DIS
LIN {X -8.264,Y 129.1932,Z 155,A 92.0733,B 16.1461,C -0.4038,E1 16.1417,E2 717.0073} C_DIS
LIN {X -5.4149,Y 129.3441,Z 155,A 90.4578,B 16.1464,C -0.393,E1 16.1463,E2 718.6623} C_DIS
LIN {X -1.2114,Y 129.4522,Z 155,A 88.6668,B 16.1464,C -0.3955,E1 16.1513,E2 720.4445} C_DIS
LIN {X 5.7204,Y 129.3312,Z 155,A 85.7672,B 16.1462,C -0.401,E1 16.1594,E2 723.3235} C_DIS
LIN {X 8.3717,Y 129.1865,Z 155,A 83.8098,B 16.1468,C -0.376,E1 16.1651,E2 725.3691} C_DIS
LIN {X 13.4559,Y 128.7562,Z 155,A 82.1081,B 16.1464,C -0.3933,E1 16.1696,E2 727.0071} C_DIS
LIN {X 17.0119,Y 128.3342,Z 155,A 80.6574,B 16.1464,C -0.3971,E1 16.1736,E2 728.4421} C_DIS
LIN {X 20.7095,Y 127.7909,Z 155,A 78.6891,B 16.1466,C -0.3864,E1 16.1791,E2 730.4456} C_DIS
LIN {X 25.1076,Y 127.0006,Z 155,A 77.0705,B 16.1463,C -0.3971,E1 16.1834,E2 732.023} C_DIS
LIN {X 28.2689,Y 126.3337,Z 155,A 75.7014,B 16.1463,C -0.3983,E1 16.1872,E2 733.3848} C_DIS
LIN {X 30.5952,Y 125.7895,Z 155,A 74.5239,B 16.1463,C -0.3938,E1 16.1904,E2 734.5759} C_DIS
LIN {X 34.0815,Y 124.892,Z 155,A 72.7653,B 16.1465,C -0.3873,E1 16.1952,E2 736.3531} C_DIS
LIN {X 38.6381,Y 123.5585,Z 155,A 70.8741,B 16.1465,C -0.3925,E1 16.2002,E2 738.2203} C_DIS
LIN {X 41.1741,Y 122.7345,Z 155,A 69.6483,B 16.1465,C -0.39,E1 16.2034,E2 739.4511} C_DIS
LIN {X 49.5902,Y 119.5821,Z 155,A 65.7815,B 16.1465,C -0.3897,E1 16.2135,E2 743.3054} C_DIS
LIN {X 53.531,Y 117.8725,Z 155,A 63.8393,B 16.1465,C -0.3862,E1 16.2185,E2 745.2524} C_DIS
LIN {X 56.742,Y 116.3599,Z 155,A 62.3511,B 16.1465,C -0.3871,E1 16.2222,E2 746.7313} C_DIS
LIN {X 59.6255,Y 114.9093,Z 155,A 60.7547,B 16.1467,C -0.3797,E1 16.2262,E2 748.3472} C_DIS
LIN {X 67.5201,Y 110.456,Z 155,A 56.9345,B 16.1467,C -0.3803,E1 16.2355,E2 752.1465} C_DIS
LIN {X 70.4512,Y 108.6097,Z 155,A 55.3997,B 16.1467,C -0.3779,E1 16.2391,E2 753.6819} C_DIS
LIN {X 73.5372,Y 106.5451,Z 155,A 53.6873,B 16.1469,C -0.3729,E1 16.243,E2 755.4029} C_DIS
LIN {X 76.578,Y 104.3804,Z 155,A 51.9009,B 16.147,C -0.3656,E1 16.2471,E2 757.2053} C_DIS
LIN {X 80.2765,Y 101.5642,Z 155,A 49.8515,B 16.1471,C -0.3622,E1 16.2516,E2 759.2547} C_DIS
LIN {X 83.5755,Y 98.8671,Z 155,A 48.084,B 16.1471,C -0.3628,E1 16.2554,E2 761.0094} C_DIS
LIN {X 86.2922,Y 96.5045,Z 155,A 46.5124,B 16.1471,C -0.3604,E1 16.2587,E2 762.5793} C_DIS
LIN {X 89.401,Y 93.6318,Z 155,A 44.5963,B 16.1473,C -0.3552,E1 16.2626,E2 764.5012} C_DIS
LIN {X 92.4343,Y 90.6386,Z 155,A 42.7053,B 16.1473,C -0.3512,E1 16.2663,E2 766.3938} C_DIS
LIN {X 95.1318,Y 87.8034,Z 155,A 40.9448,B 16.1474,C -0.3465,E1 16.2697,E2 768.1587} C_DIS
LIN {X 98.2674,Y 84.2796,Z 155,A 38.9824,B 16.1474,C -0.3462,E1 16.2733,E2 770.1081} C_DIS
LIN {X 100.8607,Y 81.1578,Z 155,A 37.2569,B 16.1474,C -0.3445,E1 16.2763,E2 771.8266} C_DIS
LIN {X 103.0106,Y 78.4114,Z 155,A 35.651,B 16.1476,C -0.3388,E1 16.2791,E2 773.4409} C_DIS
LIN {X 108.6128,Y 70.4464,Z 155,A 31.581,B 16.1476,C -0.3366,E1 16.2856,E2 777.4865} C_DIS
LIN {X 110.5389,Y 67.385,Z 155,A 29.8134,B 16.1478,C -0.3267,E1 16.2882,E2 779.2749} C_DIS
LIN {X 112.5573,Y 63.9559,Z 155,A 28.1309,B 16.1478,C -0.3249,E1 16.2905,E2 780.9498} C_DIS
LIN {X 113.8837,Y 61.5634,Z 155,A 26.8125,B 16.148,C -0.318,E1 16.2923,E2 782.2818} C_DIS
LIN {X 115.6573,Y 58.1612,Z 155,A 24.2803,B 16.1486,C -0.2846,E1 16.2956,E2 784.9114} C_DIS
LIN {X 118.331,Y 52.5059,Z 155,A 22.925,B 16.1478,C -0.3263,E1 16.297,E2 786.1061} C_DIS
LIN {X 119.7688,Y 49.143,Z 155,A 20.8543,B 16.1482,C -0.3059,E1 16.2993,E2 788.2314} C_DIS
LIN {X 121.1617,Y 45.5943,Z 155,A 19.1474,B 16.1483,C -0.3006,E1 16.3011,E2 789.9423} C_DIS
LIN {X 122.2633,Y 42.552,Z 155,A 17.7422,B 16.1483,C -0.2975,E1 16.3024,E2 791.3458} C_DIS
LIN {X 123.3426,Y 39.314,Z 155,A 16.2691,B 16.1484,C -0.2945,E1 16.3036,E2 792.8162} C_DIS
LIN {X 124.4855,Y 35.5363,Z 155,A 14.5769,B 16.1485,C -0.2913,E1 16.305,E2 794.504} C_DIS
LIN {X 125.3373,Y 32.4018,Z 155,A 12.9469,B 16.1487,C -0.2804,E1 16.3062,E2 796.158} C_DIS
LIN {X 126.6384,Y 26.869,Z 155,A 10.3826,B 16.1488,C -0.2713,E1 16.3077,E2 798.7308} C_DIS
LIN {X 127.5004,Y 22.4236,Z 155,A 8.553,B 16.1488,C -0.2715,E1 16.3087,E2 800.5424} C_DIS
LIN {X 128.2341,Y 17.7522,Z 155,A 6.375,B 16.149,C -0.2622,E1 16.3096,E2 802.7329} C_DIS
LIN {X 129.114,Y 9.4156,Z 155,A 2.8509,B 16.149,C -0.2576,E1 16.3105,E2 806.24} C_DIS
LIN {X 129.3885,Y 4.2597,Z 155,A 0.5157,B 16.1492,C -0.2489,E1 16.3108,E2 808.584} C_DIS
LIN {X 129.458,Y 0.3178,Z 155,A -1.2566,B 16.1492,C -0.2426,E1 16.3108,E2 810.3617} C_DIS
LIN {X 129.4113,Y -3.4402,Z 155,A -2.7896,B 16.1492,C -0.2422,E1 16.3108,E2 811.8815} C_DIS
Enddeposition()
END
